// TIA Portal V19 export
// export: Created 2024-12-05T09:06:09.934265Z, ExportSetting WithDefaults, DisplayName Totally Integrated Automation Portal, DisplayVersion V19 Update 1, DisplayName TIA Portal Openness, DisplayVersion V19 Update 1, DisplayName TIA Portal Version Control Interface, DisplayVersion V19, DisplayName SINAMICS Startdrive Advanced, DisplayVersion V19, DisplayName SINAMICS DCC, DisplayVersion V19, DisplayName SINAMICS Startdrive G130, G150, S120, S150, SINAMICS MV, G220, S200, S210, DisplayVersion V19, DisplayName SINAMICS Startdrive G110M, G120, G120C, G120D, G120P, G115D, DisplayVersion V19, DisplayName STEP 7 Professional, DisplayVersion V19 Update 1, DisplayName STEP 7 Safety, DisplayVersion V19 Update 1, DisplayName WinCC Advanced, DisplayVersion V19 Update 1, DisplayName WinCC Advanced / Unified PC, DisplayVersion V19 Update 1
DATA_BLOCK "CH1"   // DB7
{ S7_Optimized_Access := 'TRUE' }
VERSION : 0.1
// stored: AutoNumber true, DBAccessibleFromOPCUA true, DBAccessibleFromWebserver true, InstanceOfName CH, InstanceOfType UDT, IsOnlyStoredInLoadMemory false, IsWriteProtectedInAS false
"CH"
   // VAR RETAIN
   //    Std : "EM_Std";
   //    Gen : "CH_Gen";
   //    Param : "CH_Param";
   //    LastHmiDataParam : "CH_Param";
   //    Alm : "CH_Alm";
   //    Sign : "EM_Sign";
   //    Input : "CH_Input";
   //    Output : "CH_Output";
   //    Ons : "CH_Ons";
   //    "Step" : "CH_Step";
   //    CamCalc : "CH_CamCalc";
   //    Chain1Long : "CH_Chain";
   //    Chain2Long : "CH_Chain";
   //    Chain3Long : "CH_Chain";
   //    Chain4Cross : "CH_Chain";
   //    Chain5Long : "CH_Chain";
   //    Chain6Long : "CH_Chain";
   //    Chain7Long : "CH_Chain";
   //    Chain8Cross : "CH_Chain";
   //    VMaster : "CH_Virtual";
   //    VMasterBooked : "CH_VirtualBooked";
   // END_VAR
BEGIN
   Std.Cfg_ModuleSync := TRUE;
   Std.Cfg_0_BelongShort_1_BelongLong := TRUE;
   Std.Cfg_ExternalCPU := FALSE;
   Std.Cfg_0_JogWord_1_JogBit := TRUE;
   Std._0_PriorityAlm_1_FirstAlm := FALSE;
   Std.AbortAlmOk := TRUE;
   Std.ServicesAbortAlmOk := FALSE;
   Std.SignOK := TRUE;
   Std.AlmReset := FALSE;
   Std.SignReset := FALSE;
   Std.NewAlm := FALSE;
   Std.NewSign := FALSE;
   Std.RstNewAlm := FALSE;
   Std.RstNewSign := FALSE;
   Std.AllowCopyByCategory := TRUE;
   Std.ForceCopyAll := FALSE;
   Std.InitCategories := FALSE;
   Std.InitCauses := FALSE;
   Std.Diag_AlmFound := FALSE;
   Std.Diag_SignFound := FALSE;
   Std.ScOk := FALSE;
   Std.OkToStop := TRUE;
   Std.PwrDrv := TRUE;
   Std.DriveRunCmd := FALSE;
   Std.ManAct := FALSE;
   Std.MachineSelected := TRUE;
   Std.MachineExtracted := FALSE;
   Std.LocalAbortReq := TRUE;
   Std.CondOkToEnaStaReq := FALSE;
   Std.EnaReq := FALSE;
   Std.EnaStaReq := FALSE;
   Std.StaReq := FALSE;
   Std.ReqStart := FALSE;
   Std.ReqStop := FALSE;
   Std.ReqAbort := TRUE;
   Std.ReqExecute := FALSE;
   Std.ReqReset := FALSE;
   Std.ReqSuspend := FALSE;
   Std.ReqUnSuspend := FALSE;
   Std.StrobeDeviceDiag := FALSE;
   Std.StrobeInverterDiag := FALSE;
   Std.DeviceDiagnosticDone := FALSE;
   Std.InverterDiagnosticDone := FALSE;
   Std.RecipeOnlineLoadDone := FALSE;
   Std.RecipeOnlineSaveDone := FALSE;
   Std.RecipeOfflineLoadDone := FALSE;
   Std.RecipeOfflineSaveDone := FALSE;
   Std.LastHmiDataLoadDone := FALSE;
   Std.LastHmiDataSaveDone := FALSE;
   Std.SummAlmTimeoutStart := FALSE;
   Std.SirenEna := FALSE;
   Std.VisEnButtons := TRUE;
   Std.VisManButtons := FALSE;
   Std.VisHomeButtons := FALSE;
   Std.VisEnButtonsRunning := TRUE;
   Std.Ena_Suspended := TRUE;
   Std.BluStkLgh_Steady_Cond := FALSE;
   Std.BluStkLgh_Frequency1_Cond := FALSE;
   Std.Siren_Frequency4_Cond := FALSE;
   Std.Cfg_ModuleNumber := 0;
   Std.Cfg_DeviceDiagCounter_Preset := 0;
   Std.Cfg_InverterDiagCounter_Preset := 0;
   Std.Cfg_Num_AlmDint := 19;
   Std.Cfg_Num_SignDint := 3;
   Std.Cfg_StaPbt := 65535;
   Std.Cfg_StoPbt := 65535;
   Std.Cfg_RstPbt := -1;
   Std.Cfg_EnaPbt := 65535;
   Std.Cfg_Siren := 1;
   Std.Cfg_Stack := 1;
   Std.Cfg_DisableStates[0..31] := 0;
   Std.Cfg_ModeTransitions[0..31] := 0;
   Std.Cfg_ModeNames[0..31] := '';
   Std.ModeCurrentName := 'Production';
   Std.StateCurrentName := 'Aborted';
   Std.DeviceDiagCounter := 0;
   Std.InverterDiagCounter := 0;
   Std.MaintenanceActivated."0" := FALSE;
   Std.MaintenanceActivated."1" := FALSE;
   Std.MaintenanceActivated."2" := FALSE;
   Std.MaintenanceActivated."3" := FALSE;
   Std.MaintenanceActivated."4" := FALSE;
   Std.MaintenanceActivated."5" := FALSE;
   Std.MaintenanceActivated."6" := FALSE;
   Std.MaintenanceActivated."7" := FALSE;
   Std.MaintenanceActivated."8" := FALSE;
   Std.MaintenanceActivated."9" := FALSE;
   Std.MaintenanceActivated."10" := FALSE;
   Std.MaintenanceActivated."11" := FALSE;
   Std.MaintenanceActivated."12" := FALSE;
   Std.MaintenanceActivated."13" := FALSE;
   Std.MaintenanceActivated."14" := FALSE;
   Std.MaintenanceActivated."15" := FALSE;
   Std.MaintenanceActivated."16" := FALSE;
   Std.MaintenanceActivated."17" := FALSE;
   Std.MaintenanceActivated."18" := FALSE;
   Std.MaintenanceActivated."19" := FALSE;
   Std.MaintenanceActivated."20" := FALSE;
   Std.MaintenanceActivated."21" := FALSE;
   Std.MaintenanceActivated."22" := FALSE;
   Std.MaintenanceActivated."23" := FALSE;
   Std.MaintenanceActivated."24" := FALSE;
   Std.MaintenanceActivated."25" := FALSE;
   Std.MaintenanceActivated."26" := FALSE;
   Std.MaintenanceActivated."27" := FALSE;
   Std.MaintenanceActivated."28" := FALSE;
   Std.MaintenanceActivated."29" := FALSE;
   Std.MaintenanceActivated."30" := FALSE;
   Std.MaintenanceActivated."31" := FALSE;
   Std.MaintenanceReq."0" := FALSE;
   Std.MaintenanceReq."1" := FALSE;
   Std.MaintenanceReq."2" := FALSE;
   Std.MaintenanceReq."3" := FALSE;
   Std.MaintenanceReq."4" := FALSE;
   Std.MaintenanceReq."5" := FALSE;
   Std.MaintenanceReq."6" := FALSE;
   Std.MaintenanceReq."7" := FALSE;
   Std.MaintenanceReq."8" := FALSE;
   Std.MaintenanceReq."9" := FALSE;
   Std.MaintenanceReq."10" := FALSE;
   Std.MaintenanceReq."11" := FALSE;
   Std.MaintenanceReq."12" := FALSE;
   Std.MaintenanceReq."13" := FALSE;
   Std.MaintenanceReq."14" := FALSE;
   Std.MaintenanceReq."15" := FALSE;
   Std.MaintenanceReq."16" := FALSE;
   Std.MaintenanceReq."17" := FALSE;
   Std.MaintenanceReq."18" := FALSE;
   Std.MaintenanceReq."19" := FALSE;
   Std.MaintenanceReq."20" := FALSE;
   Std.MaintenanceReq."21" := FALSE;
   Std.MaintenanceReq."22" := FALSE;
   Std.MaintenanceReq."23" := FALSE;
   Std.MaintenanceReq."24" := FALSE;
   Std.MaintenanceReq."25" := FALSE;
   Std.MaintenanceReq."26" := FALSE;
   Std.MaintenanceReq."27" := FALSE;
   Std.MaintenanceReq."28" := FALSE;
   Std.MaintenanceReq."29" := FALSE;
   Std.MaintenanceReq."30" := FALSE;
   Std.MaintenanceReq."31" := FALSE;
   Std.WithinScreenRange := 0;
   Std.ExchangeToGlobal.Communication.RunMode := FALSE;
   Std.ExchangeToGlobal.Communication.ConnectionFaulted := FALSE;
   Std.ExchangeToGlobal.Gen.Communication := FALSE;
   Std.ExchangeToGlobal.Gen.Selected := TRUE;
   Std.ExchangeToGlobal.Gen.Extracted := FALSE;
   Std.ExchangeToGlobal.Gen.EnaReq := FALSE;
   Std.ExchangeToGlobal.Gen.StaReq := FALSE;
   Std.ExchangeToGlobal.Gen.Started := FALSE;
   Std.ExchangeToGlobal.Gen.Unsuspended := FALSE;
   Std.ExchangeToGlobal.Gen.Ena_Suspended := TRUE;
   Std.ExchangeToGlobal.Gen.sts_Starting := FALSE;
   Std.ExchangeToGlobal.Gen.sts_Stopping := FALSE;
   Std.ExchangeToGlobal.Gen.sts_Aborting := FALSE;
   Std.ExchangeToGlobal.Gen.sts_Suspending := FALSE;
   Std.ExchangeToGlobal.Gen.sts_Unsuspending := FALSE;
   Std.ExchangeToGlobal.Gen.sts_Execute := FALSE;
   Std.ExchangeToGlobal.Gen.sts_Idle := FALSE;
   Std.ExchangeToGlobal.Gen.sts_Stopped := FALSE;
   Std.ExchangeToGlobal.Gen.sts_Aborted := TRUE;
   Std.ExchangeToGlobal.Gen.sts_Suspended := FALSE;
   Std.ExchangeToGlobal.Gen.sts_ModeManual := FALSE;
   Std.ExchangeToGlobal.Gen.sts_ModeAutomatic := TRUE;
   Std.ExchangeToGlobal.Gen.NewAlm := FALSE;
   Std.ExchangeToGlobal.Gen.NewSign := FALSE;
   Std.ExchangeToGlobal.Gen.RecipeOnlineLoadDone := FALSE;
   Std.ExchangeToGlobal.Gen.RecipeOnlineSaveDone := FALSE;
   Std.ExchangeToGlobal.Gen.RecipeOfflineLoadDone := FALSE;
   Std.ExchangeToGlobal.Gen.RecipeOfflineSaveDone := FALSE;
   Std.ExchangeToGlobal.Gen.LastHmiDataLoadDone := FALSE;
   Std.ExchangeToGlobal.Gen.LastHmiDataSaveDone := FALSE;
   Std.ExchangeToGlobal.Gen.InverterDiagnosticDone := FALSE;
   Std.ExchangeToGlobal.Gen.AxisGroupSync := TRUE;
   Std.ExchangeToGlobal.Gen.CmdMode := 1;
   Std.ExchangeToGlobal.Gen.Mode := 1;
   Std.ExchangeToGlobal.Gen.DisableEnaPbt := 0;
   Std.ExchangeToGlobal.Input.StaPbt := FALSE;
   Std.ExchangeToGlobal.Input.StoPbt := FALSE;
   Std.ExchangeToGlobal.Input.RstPbt := FALSE;
   Std.ExchangeToGlobal.Input.EnaPbt := FALSE;
   Std.ExchangeToGlobal.Input._4 := FALSE;
   Std.ExchangeToGlobal.Input._5 := FALSE;
   Std.ExchangeToGlobal.Input._6 := FALSE;
   Std.ExchangeToGlobal.Input._7 := FALSE;
   Std.ExchangeToGlobal.Input._8 := FALSE;
   Std.ExchangeToGlobal.Input._9 := FALSE;
   Std.ExchangeToGlobal.Input._10 := FALSE;
   Std.ExchangeToGlobal.Input._11 := FALSE;
   Std.ExchangeToGlobal.Input._12 := FALSE;
   Std.ExchangeToGlobal.Input._13 := FALSE;
   Std.ExchangeToGlobal.Input._14 := FALSE;
   Std.ExchangeToGlobal.Input._15 := FALSE;
   Std.ExchangeToGlobal.AlmOk.ThSwitch := TRUE;
   Std.ExchangeToGlobal.AlmOk.SafeComm := TRUE;
   Std.ExchangeToGlobal.AlmOk.SafeEmg := TRUE;
   Std.ExchangeToGlobal.AlmOk.SafeGuards := TRUE;
   Std.ExchangeToGlobal.AlmOk.GtaAirGroup := TRUE;
   Std.ExchangeToGlobal.AlmOk.Major := TRUE;
   Std.ExchangeToGlobal.AlmOk.Minor := TRUE;
   Std.ExchangeToGlobal.AlmOk.Spare07 := TRUE;
   Std.ExchangeToGlobal.AlmOk.Spare08 := TRUE;
   Std.ExchangeToGlobal.AlmOk.Spare09 := TRUE;
   Std.ExchangeToGlobal.AlmOk.Spare10 := TRUE;
   Std.ExchangeToGlobal.AlmOk.Spare11 := TRUE;
   Std.ExchangeToGlobal.AlmOk.Spare12 := TRUE;
   Std.ExchangeToGlobal.AlmOk.Spare13 := TRUE;
   Std.ExchangeToGlobal.AlmOk.Spare14 := TRUE;
   Std.ExchangeToGlobal.AlmOk.Spare15 := TRUE;
   Std.ExchangeToGlobal.AlmOk.Spare16 := TRUE;
   Std.ExchangeToGlobal.AlmOk.Spare17 := TRUE;
   Std.ExchangeToGlobal.AlmOk.Spare18 := TRUE;
   Std.ExchangeToGlobal.AlmOk.Spare19 := TRUE;
   Std.ExchangeToGlobal.AlmOk.Spare20 := TRUE;
   Std.ExchangeToGlobal.AlmOk.Spare21 := TRUE;
   Std.ExchangeToGlobal.AlmOk.Spare22 := TRUE;
   Std.ExchangeToGlobal.AlmOk.Spare23 := TRUE;
   Std.ExchangeToGlobal.AlmOk.Spare24 := TRUE;
   Std.ExchangeToGlobal.AlmOk.Spare25 := TRUE;
   Std.ExchangeToGlobal.AlmOk.Spare26 := TRUE;
   Std.ExchangeToGlobal.AlmOk.Spare27 := TRUE;
   Std.ExchangeToGlobal.AlmOk.Spare28 := TRUE;
   Std.ExchangeToGlobal.AlmOk.Spare29 := TRUE;
   Std.ExchangeToGlobal.AlmOk.Spare30 := TRUE;
   Std.ExchangeToGlobal.AlmOk.Spare31 := TRUE;
   Std.ExchangeToGlobal.AlmCauseOk.Ope := TRUE;
   Std.ExchangeToGlobal.AlmCauseOk.Ust := TRUE;
   Std.ExchangeToGlobal.AlmCauseOk.Dst := TRUE;
   Std.ExchangeToGlobal.AlmCauseOk.Ext := TRUE;
   Std.ExchangeToGlobal.AlmCauseOk.Mac := TRUE;
   Std.ExchangeToGlobal.AlmCauseOk.Spare05 := TRUE;
   Std.ExchangeToGlobal.AlmCauseOk.Spare06 := TRUE;
   Std.ExchangeToGlobal.AlmCauseOk.Spare07 := TRUE;
   Std.ExchangeToGlobal.AlmCauseOk.Spare08 := TRUE;
   Std.ExchangeToGlobal.AlmCauseOk.Spare09 := TRUE;
   Std.ExchangeToGlobal.AlmCauseOk.Spare10 := TRUE;
   Std.ExchangeToGlobal.AlmCauseOk.Spare11 := TRUE;
   Std.ExchangeToGlobal.AlmCauseOk.Spare12 := TRUE;
   Std.ExchangeToGlobal.AlmCauseOk.Spare13 := TRUE;
   Std.ExchangeToGlobal.AlmCauseOk.Spare14 := TRUE;
   Std.ExchangeToGlobal.AlmCauseOk.Spare15 := TRUE;
   Std.ExchangeToGlobal.AlmCauseOk.Spare16 := TRUE;
   Std.ExchangeToGlobal.AlmCauseOk.Spare17 := TRUE;
   Std.ExchangeToGlobal.AlmCauseOk.Spare18 := TRUE;
   Std.ExchangeToGlobal.AlmCauseOk.Spare19 := TRUE;
   Std.ExchangeToGlobal.AlmCauseOk.Spare20 := TRUE;
   Std.ExchangeToGlobal.AlmCauseOk.Spare21 := TRUE;
   Std.ExchangeToGlobal.AlmCauseOk.Spare22 := TRUE;
   Std.ExchangeToGlobal.AlmCauseOk.Spare23 := TRUE;
   Std.ExchangeToGlobal.AlmCauseOk.Spare24 := TRUE;
   Std.ExchangeToGlobal.AlmCauseOk.Spare25 := TRUE;
   Std.ExchangeToGlobal.AlmCauseOk.Spare26 := TRUE;
   Std.ExchangeToGlobal.AlmCauseOk.Spare27 := TRUE;
   Std.ExchangeToGlobal.AlmCauseOk.Spare28 := TRUE;
   Std.ExchangeToGlobal.AlmCauseOk.Spare29 := TRUE;
   Std.ExchangeToGlobal.AlmCauseOk.Spare30 := TRUE;
   Std.ExchangeToGlobal.AlmCauseOk.Spare31 := TRUE;
   Std.ExchangeToGlobal.AlmBannerFbk.FirstAlmDetection := FALSE;
   Std.ExchangeToGlobal.AlmBannerFbk.AlmPriority := 100;
   Std.ExchangeToGlobal.AlmBannerFbk.AlmCategory := -1;
   Std.ExchangeToGlobal.AlmBannerFbk.AlmCause := -1;
   Std.ExchangeToGlobal.AlmBannerFbk.AlmID := -1;
   Std.ExchangeToGlobal.AlmBannerFbk.GlobalAbsTime := 0;
   Std.ExchangeToGlobal.SignBannerFbk.SignPriority := 100;
   Std.ExchangeToGlobal.SignBannerFbk.SignCategory := -1;
   Std.ExchangeToGlobal.SignBannerFbk.SignID := -1;
   Std.ExchangeToGlobal.ExtCPU.PushButton.StaPbt := FALSE;
   Std.ExchangeToGlobal.ExtCPU.PushButton.StoPbt := FALSE;
   Std.ExchangeToGlobal.ExtCPU.PushButton.RstPbt := FALSE;
   Std.ExchangeToGlobal.ExtCPU.PushButton.EnaPbt := FALSE;
   Std.ExchangeToGlobal.ExtCPU.PushButton.EnaReq := FALSE;
   Std.ExchangeToGlobal.ExtCPU.PushButton.EnaStaReq := FALSE;
   Std.ExchangeToGlobal.ExtCPU.DeviceDiagDone := FALSE;
   Std.ExchangeToGlobal.ExtCPU.InverterDiagDone := FALSE;
   Std.ExchangeToGlobal.LightSiren.Cfg_StaPbt := 65535;
   Std.ExchangeToGlobal.LightSiren.Cfg_RstPbt := -1;
   Std.ExchangeToGlobal.LightSiren.Cfg_EnaPbt := 65535;
   Std.ExchangeToGlobal.LightSiren.Cfg_Siren := 1;
   Std.ExchangeToGlobal.LightSiren.Cfg_Stack := 1;
   Std.ExchangeToGlobal.LightSiren.Steady.StaPbtLgh := FALSE;
   Std.ExchangeToGlobal.LightSiren.Steady.RstPbtLgh := FALSE;
   Std.ExchangeToGlobal.LightSiren.Steady.EnaPbtLgh := FALSE;
   Std.ExchangeToGlobal.LightSiren.Steady.Siren := FALSE;
   Std.ExchangeToGlobal.LightSiren.Steady.YelStkLgh := FALSE;
   Std.ExchangeToGlobal.LightSiren.Steady.BluStkLgh := FALSE;
   Std.ExchangeToGlobal.LightSiren.Steady.GrnStkLgh := FALSE;
   Std.ExchangeToGlobal.LightSiren.Steady.WhtStkLgh := FALSE;
   Std.ExchangeToGlobal.LightSiren.Steady.Cust1_StaPbtLgh := FALSE;
   Std.ExchangeToGlobal.LightSiren.Steady.Cust1_RstPbtLgh := FALSE;
   Std.ExchangeToGlobal.LightSiren.Steady.Cust1_Siren := FALSE;
   Std.ExchangeToGlobal.LightSiren.Steady.Cust1_RedStkLgh := FALSE;
   Std.ExchangeToGlobal.LightSiren.Steady.Cust1_OngStkLgh := FALSE;
   Std.ExchangeToGlobal.LightSiren.Steady.Cust1_GrnStkLgh := FALSE;
   Std.ExchangeToGlobal.LightSiren.Steady.Cust1_BluStkLgh := FALSE;
   Std.ExchangeToGlobal.LightSiren.Steady.Cust1_WhtStkLgh := FALSE;
   Std.ExchangeToGlobal.LightSiren.Frequency1.StaPbtLgh := FALSE;
   Std.ExchangeToGlobal.LightSiren.Frequency1.RstPbtLgh := FALSE;
   Std.ExchangeToGlobal.LightSiren.Frequency1.EnaPbtLgh := FALSE;
   Std.ExchangeToGlobal.LightSiren.Frequency1.Siren := FALSE;
   Std.ExchangeToGlobal.LightSiren.Frequency1.YelStkLgh := FALSE;
   Std.ExchangeToGlobal.LightSiren.Frequency1.BluStkLgh := FALSE;
   Std.ExchangeToGlobal.LightSiren.Frequency1.GrnStkLgh := FALSE;
   Std.ExchangeToGlobal.LightSiren.Frequency1.WhtStkLgh := FALSE;
   Std.ExchangeToGlobal.LightSiren.Frequency1.Cust1_StaPbtLgh := FALSE;
   Std.ExchangeToGlobal.LightSiren.Frequency1.Cust1_RstPbtLgh := FALSE;
   Std.ExchangeToGlobal.LightSiren.Frequency1.Cust1_Siren := FALSE;
   Std.ExchangeToGlobal.LightSiren.Frequency1.Cust1_RedStkLgh := FALSE;
   Std.ExchangeToGlobal.LightSiren.Frequency1.Cust1_OngStkLgh := FALSE;
   Std.ExchangeToGlobal.LightSiren.Frequency1.Cust1_GrnStkLgh := FALSE;
   Std.ExchangeToGlobal.LightSiren.Frequency1.Cust1_BluStkLgh := FALSE;
   Std.ExchangeToGlobal.LightSiren.Frequency1.Cust1_WhtStkLgh := FALSE;
   Std.ExchangeToGlobal.LightSiren.Frequency2.StaPbtLgh := FALSE;
   Std.ExchangeToGlobal.LightSiren.Frequency2.RstPbtLgh := FALSE;
   Std.ExchangeToGlobal.LightSiren.Frequency2.EnaPbtLgh := FALSE;
   Std.ExchangeToGlobal.LightSiren.Frequency2.Siren := FALSE;
   Std.ExchangeToGlobal.LightSiren.Frequency2.YelStkLgh := FALSE;
   Std.ExchangeToGlobal.LightSiren.Frequency2.BluStkLgh := FALSE;
   Std.ExchangeToGlobal.LightSiren.Frequency2.GrnStkLgh := FALSE;
   Std.ExchangeToGlobal.LightSiren.Frequency2.WhtStkLgh := FALSE;
   Std.ExchangeToGlobal.LightSiren.Frequency2.Cust1_StaPbtLgh := FALSE;
   Std.ExchangeToGlobal.LightSiren.Frequency2.Cust1_RstPbtLgh := FALSE;
   Std.ExchangeToGlobal.LightSiren.Frequency2.Cust1_Siren := FALSE;
   Std.ExchangeToGlobal.LightSiren.Frequency2.Cust1_RedStkLgh := FALSE;
   Std.ExchangeToGlobal.LightSiren.Frequency2.Cust1_OngStkLgh := FALSE;
   Std.ExchangeToGlobal.LightSiren.Frequency2.Cust1_GrnStkLgh := FALSE;
   Std.ExchangeToGlobal.LightSiren.Frequency2.Cust1_BluStkLgh := FALSE;
   Std.ExchangeToGlobal.LightSiren.Frequency2.Cust1_WhtStkLgh := FALSE;
   Std.ExchangeToGlobal.LightSiren.Frequency3.StaPbtLgh := FALSE;
   Std.ExchangeToGlobal.LightSiren.Frequency3.RstPbtLgh := FALSE;
   Std.ExchangeToGlobal.LightSiren.Frequency3.EnaPbtLgh := FALSE;
   Std.ExchangeToGlobal.LightSiren.Frequency3.Siren := FALSE;
   Std.ExchangeToGlobal.LightSiren.Frequency3.YelStkLgh := FALSE;
   Std.ExchangeToGlobal.LightSiren.Frequency3.BluStkLgh := FALSE;
   Std.ExchangeToGlobal.LightSiren.Frequency3.GrnStkLgh := FALSE;
   Std.ExchangeToGlobal.LightSiren.Frequency3.WhtStkLgh := FALSE;
   Std.ExchangeToGlobal.LightSiren.Frequency3.Cust1_StaPbtLgh := FALSE;
   Std.ExchangeToGlobal.LightSiren.Frequency3.Cust1_RstPbtLgh := FALSE;
   Std.ExchangeToGlobal.LightSiren.Frequency3.Cust1_Siren := FALSE;
   Std.ExchangeToGlobal.LightSiren.Frequency3.Cust1_RedStkLgh := FALSE;
   Std.ExchangeToGlobal.LightSiren.Frequency3.Cust1_OngStkLgh := FALSE;
   Std.ExchangeToGlobal.LightSiren.Frequency3.Cust1_GrnStkLgh := FALSE;
   Std.ExchangeToGlobal.LightSiren.Frequency3.Cust1_BluStkLgh := FALSE;
   Std.ExchangeToGlobal.LightSiren.Frequency3.Cust1_WhtStkLgh := FALSE;
   Std.ExchangeToGlobal.LightSiren.Frequency4.StaPbtLgh := FALSE;
   Std.ExchangeToGlobal.LightSiren.Frequency4.RstPbtLgh := FALSE;
   Std.ExchangeToGlobal.LightSiren.Frequency4.EnaPbtLgh := FALSE;
   Std.ExchangeToGlobal.LightSiren.Frequency4.Siren := FALSE;
   Std.ExchangeToGlobal.LightSiren.Frequency4.YelStkLgh := FALSE;
   Std.ExchangeToGlobal.LightSiren.Frequency4.BluStkLgh := FALSE;
   Std.ExchangeToGlobal.LightSiren.Frequency4.GrnStkLgh := FALSE;
   Std.ExchangeToGlobal.LightSiren.Frequency4.WhtStkLgh := FALSE;
   Std.ExchangeToGlobal.LightSiren.Frequency4.Cust1_StaPbtLgh := FALSE;
   Std.ExchangeToGlobal.LightSiren.Frequency4.Cust1_RstPbtLgh := FALSE;
   Std.ExchangeToGlobal.LightSiren.Frequency4.Cust1_Siren := FALSE;
   Std.ExchangeToGlobal.LightSiren.Frequency4.Cust1_RedStkLgh := FALSE;
   Std.ExchangeToGlobal.LightSiren.Frequency4.Cust1_OngStkLgh := FALSE;
   Std.ExchangeToGlobal.LightSiren.Frequency4.Cust1_GrnStkLgh := FALSE;
   Std.ExchangeToGlobal.LightSiren.Frequency4.Cust1_BluStkLgh := FALSE;
   Std.ExchangeToGlobal.LightSiren.Frequency4.Cust1_WhtStkLgh := FALSE;
   Std.ExchangeToGlobal.PackML.Sts_Aborted := TRUE;
   Std.ExchangeToGlobal.PackML.Sts_Aborting := FALSE;
   Std.ExchangeToGlobal.PackML.Sts_Clearing := FALSE;
   Std.ExchangeToGlobal.PackML.Sts_Complete := FALSE;
   Std.ExchangeToGlobal.PackML.Sts_Completing := FALSE;
   Std.ExchangeToGlobal.PackML.Sts_Execute := FALSE;
   Std.ExchangeToGlobal.PackML.Sts_Held := FALSE;
   Std.ExchangeToGlobal.PackML.Sts_Holding := FALSE;
   Std.ExchangeToGlobal.PackML.Sts_Idle := FALSE;
   Std.ExchangeToGlobal.PackML.Sts_Resetting := FALSE;
   Std.ExchangeToGlobal.PackML.Sts_Starting := FALSE;
   Std.ExchangeToGlobal.PackML.Sts_Stopped := FALSE;
   Std.ExchangeToGlobal.PackML.Sts_Stopping := FALSE;
   Std.ExchangeToGlobal.PackML.Sts_Suspended := FALSE;
   Std.ExchangeToGlobal.PackML.Sts_Suspending := FALSE;
   Std.ExchangeToGlobal.PackML.Sts_UnHolding := FALSE;
   Std.ExchangeToGlobal.PackML.Sts_UnSuspending := FALSE;
   Std.ExchangeToGlobal.PackML.Sts_AbortedEnabled := TRUE;
   Std.ExchangeToGlobal.PackML.Sts_AbortingEnabled := TRUE;
   Std.ExchangeToGlobal.PackML.Sts_ClearingEnabled := TRUE;
   Std.ExchangeToGlobal.PackML.Sts_CompleteEnabled := FALSE;
   Std.ExchangeToGlobal.PackML.Sts_CompletingEnabled := FALSE;
   Std.ExchangeToGlobal.PackML.Sts_ExecuteEnabled := TRUE;
   Std.ExchangeToGlobal.PackML.Sts_HeldEnabled := FALSE;
   Std.ExchangeToGlobal.PackML.Sts_HoldingEnabled := FALSE;
   Std.ExchangeToGlobal.PackML.Sts_IdleEnabled := TRUE;
   Std.ExchangeToGlobal.PackML.Sts_ResettingEnabled := TRUE;
   Std.ExchangeToGlobal.PackML.Sts_StartingEnabled := TRUE;
   Std.ExchangeToGlobal.PackML.Sts_StoppedEnabled := TRUE;
   Std.ExchangeToGlobal.PackML.Sts_StoppingEnabled := TRUE;
   Std.ExchangeToGlobal.PackML.Sts_SuspendedEnabled := TRUE;
   Std.ExchangeToGlobal.PackML.Sts_SuspendingEnabled := TRUE;
   Std.ExchangeToGlobal.PackML.Sts_UnHoldingEnabled := FALSE;
   Std.ExchangeToGlobal.PackML.Sts_UnSuspendingEnabled := TRUE;
   Std.ExchangeToGlobal.SignOk := TRUE;
   Std.ExchangeToGlobal."Dint"[0..4] := 0;
   Std.VisAlmTypeBool.ThSwitch := FALSE;
   Std.VisAlmTypeBool.SafeComm := FALSE;
   Std.VisAlmTypeBool.SafeEmg := FALSE;
   Std.VisAlmTypeBool.SafeGuards := TRUE;
   Std.VisAlmTypeBool.GtaAirGroup := FALSE;
   Std.VisAlmTypeBool.Major := FALSE;
   Std.VisAlmTypeBool.Minor := FALSE;
   Std.VisAlmTypeBool.Spare07 := FALSE;
   Std.VisAlmTypeBool.Spare08 := FALSE;
   Std.VisAlmTypeBool.Spare09 := FALSE;
   Std.VisAlmTypeBool.Spare10 := FALSE;
   Std.VisAlmTypeBool.Spare11 := FALSE;
   Std.VisAlmTypeBool.Spare12 := FALSE;
   Std.VisAlmTypeBool.Spare13 := FALSE;
   Std.VisAlmTypeBool.Spare14 := FALSE;
   Std.VisAlmTypeBool.Spare15 := FALSE;
   Std.VisAlmTypeBool.Spare16 := FALSE;
   Std.VisAlmTypeBool.Spare17 := FALSE;
   Std.VisAlmTypeBool.Spare18 := FALSE;
   Std.VisAlmTypeBool.Spare19 := FALSE;
   Std.VisAlmTypeBool.Spare20 := FALSE;
   Std.VisAlmTypeBool.Spare21 := FALSE;
   Std.VisAlmTypeBool.Spare22 := FALSE;
   Std.VisAlmTypeBool.Spare23 := FALSE;
   Std.VisAlmTypeBool.Spare24 := FALSE;
   Std.VisAlmTypeBool.Spare25 := FALSE;
   Std.VisAlmTypeBool.Spare26 := FALSE;
   Std.VisAlmTypeBool.Spare27 := FALSE;
   Std.VisAlmTypeBool.Spare28 := FALSE;
   Std.VisAlmTypeBool.Spare29 := FALSE;
   Std.VisAlmTypeBool.Spare30 := FALSE;
   Std.VisAlmTypeBool.Spare31 := FALSE;
   Std.AlmTypeFbk.ThSwitch := FALSE;
   Std.AlmTypeFbk.SafeComm := FALSE;
   Std.AlmTypeFbk.SafeEmg := FALSE;
   Std.AlmTypeFbk.SafeGuards := FALSE;
   Std.AlmTypeFbk.GtaAirGroup := FALSE;
   Std.AlmTypeFbk.Major := FALSE;
   Std.AlmTypeFbk.Minor := FALSE;
   Std.AlmTypeFbk.Spare07 := FALSE;
   Std.AlmTypeFbk.Spare08 := FALSE;
   Std.AlmTypeFbk.Spare09 := FALSE;
   Std.AlmTypeFbk.Spare10 := FALSE;
   Std.AlmTypeFbk.Spare11 := FALSE;
   Std.AlmTypeFbk.Spare12 := FALSE;
   Std.AlmTypeFbk.Spare13 := FALSE;
   Std.AlmTypeFbk.Spare14 := FALSE;
   Std.AlmTypeFbk.Spare15 := FALSE;
   Std.AlmTypeFbk.Spare16 := FALSE;
   Std.AlmTypeFbk.Spare17 := FALSE;
   Std.AlmTypeFbk.Spare18 := FALSE;
   Std.AlmTypeFbk.Spare19 := FALSE;
   Std.AlmTypeFbk.Spare20 := FALSE;
   Std.AlmTypeFbk.Spare21 := FALSE;
   Std.AlmTypeFbk.Spare22 := FALSE;
   Std.AlmTypeFbk.Spare23 := FALSE;
   Std.AlmTypeFbk.Spare24 := FALSE;
   Std.AlmTypeFbk.Spare25 := FALSE;
   Std.AlmTypeFbk.Spare26 := FALSE;
   Std.AlmTypeFbk.Spare27 := FALSE;
   Std.AlmTypeFbk.Spare28 := FALSE;
   Std.AlmTypeFbk.Spare29 := FALSE;
   Std.AlmTypeFbk.Spare30 := FALSE;
   Std.AlmTypeFbk.Spare31 := FALSE;
   Std.AlmTypeOk.ThSwitch := TRUE;
   Std.AlmTypeOk.SafeComm := TRUE;
   Std.AlmTypeOk.SafeEmg := TRUE;
   Std.AlmTypeOk.SafeGuards := TRUE;
   Std.AlmTypeOk.GtaAirGroup := TRUE;
   Std.AlmTypeOk.Major := TRUE;
   Std.AlmTypeOk.Minor := TRUE;
   Std.AlmTypeOk.Spare07 := TRUE;
   Std.AlmTypeOk.Spare08 := TRUE;
   Std.AlmTypeOk.Spare09 := TRUE;
   Std.AlmTypeOk.Spare10 := TRUE;
   Std.AlmTypeOk.Spare11 := TRUE;
   Std.AlmTypeOk.Spare12 := TRUE;
   Std.AlmTypeOk.Spare13 := TRUE;
   Std.AlmTypeOk.Spare14 := TRUE;
   Std.AlmTypeOk.Spare15 := TRUE;
   Std.AlmTypeOk.Spare16 := TRUE;
   Std.AlmTypeOk.Spare17 := TRUE;
   Std.AlmTypeOk.Spare18 := TRUE;
   Std.AlmTypeOk.Spare19 := TRUE;
   Std.AlmTypeOk.Spare20 := TRUE;
   Std.AlmTypeOk.Spare21 := TRUE;
   Std.AlmTypeOk.Spare22 := TRUE;
   Std.AlmTypeOk.Spare23 := TRUE;
   Std.AlmTypeOk.Spare24 := TRUE;
   Std.AlmTypeOk.Spare25 := TRUE;
   Std.AlmTypeOk.Spare26 := TRUE;
   Std.AlmTypeOk.Spare27 := TRUE;
   Std.AlmTypeOk.Spare28 := TRUE;
   Std.AlmTypeOk.Spare29 := TRUE;
   Std.AlmTypeOk.Spare30 := TRUE;
   Std.AlmTypeOk.Spare31 := TRUE;
   Std.AlmCauseFbk.Ope := FALSE;
   Std.AlmCauseFbk.Ust := FALSE;
   Std.AlmCauseFbk.Dst := FALSE;
   Std.AlmCauseFbk.Ext := FALSE;
   Std.AlmCauseFbk.Mac := FALSE;
   Std.AlmCauseFbk.Spare05 := FALSE;
   Std.AlmCauseFbk.Spare06 := FALSE;
   Std.AlmCauseFbk.Spare07 := FALSE;
   Std.AlmCauseFbk.Spare08 := FALSE;
   Std.AlmCauseFbk.Spare09 := FALSE;
   Std.AlmCauseFbk.Spare10 := FALSE;
   Std.AlmCauseFbk.Spare11 := FALSE;
   Std.AlmCauseFbk.Spare12 := FALSE;
   Std.AlmCauseFbk.Spare13 := FALSE;
   Std.AlmCauseFbk.Spare14 := FALSE;
   Std.AlmCauseFbk.Spare15 := FALSE;
   Std.AlmCauseFbk.Spare16 := FALSE;
   Std.AlmCauseFbk.Spare17 := FALSE;
   Std.AlmCauseFbk.Spare18 := FALSE;
   Std.AlmCauseFbk.Spare19 := FALSE;
   Std.AlmCauseFbk.Spare20 := FALSE;
   Std.AlmCauseFbk.Spare21 := FALSE;
   Std.AlmCauseFbk.Spare22 := FALSE;
   Std.AlmCauseFbk.Spare23 := FALSE;
   Std.AlmCauseFbk.Spare24 := FALSE;
   Std.AlmCauseFbk.Spare25 := FALSE;
   Std.AlmCauseFbk.Spare26 := FALSE;
   Std.AlmCauseFbk.Spare27 := FALSE;
   Std.AlmCauseFbk.Spare28 := FALSE;
   Std.AlmCauseFbk.Spare29 := FALSE;
   Std.AlmCauseFbk.Spare30 := FALSE;
   Std.AlmCauseFbk.Spare31 := FALSE;
   Std.AlmCauseOk.Ope := TRUE;
   Std.AlmCauseOk.Ust := TRUE;
   Std.AlmCauseOk.Dst := TRUE;
   Std.AlmCauseOk.Ext := TRUE;
   Std.AlmCauseOk.Mac := TRUE;
   Std.AlmCauseOk.Spare05 := TRUE;
   Std.AlmCauseOk.Spare06 := TRUE;
   Std.AlmCauseOk.Spare07 := TRUE;
   Std.AlmCauseOk.Spare08 := TRUE;
   Std.AlmCauseOk.Spare09 := TRUE;
   Std.AlmCauseOk.Spare10 := TRUE;
   Std.AlmCauseOk.Spare11 := TRUE;
   Std.AlmCauseOk.Spare12 := TRUE;
   Std.AlmCauseOk.Spare13 := TRUE;
   Std.AlmCauseOk.Spare14 := TRUE;
   Std.AlmCauseOk.Spare15 := TRUE;
   Std.AlmCauseOk.Spare16 := TRUE;
   Std.AlmCauseOk.Spare17 := TRUE;
   Std.AlmCauseOk.Spare18 := TRUE;
   Std.AlmCauseOk.Spare19 := TRUE;
   Std.AlmCauseOk.Spare20 := TRUE;
   Std.AlmCauseOk.Spare21 := TRUE;
   Std.AlmCauseOk.Spare22 := TRUE;
   Std.AlmCauseOk.Spare23 := TRUE;
   Std.AlmCauseOk.Spare24 := TRUE;
   Std.AlmCauseOk.Spare25 := TRUE;
   Std.AlmCauseOk.Spare26 := TRUE;
   Std.AlmCauseOk.Spare27 := TRUE;
   Std.AlmCauseOk.Spare28 := TRUE;
   Std.AlmCauseOk.Spare29 := TRUE;
   Std.AlmCauseOk.Spare30 := TRUE;
   Std.AlmCauseOk.Spare31 := TRUE;
   Std.ForceCategory.ThSwitch := FALSE;
   Std.ForceCategory.SafeComm := TRUE;
   Std.ForceCategory.SafeEmg := TRUE;
   Std.ForceCategory.SafeGuards := FALSE;
   Std.ForceCategory.GtaAirGroup := FALSE;
   Std.ForceCategory.Major := FALSE;
   Std.ForceCategory.Minor := FALSE;
   Std.ForceCategory.Spare07 := FALSE;
   Std.ForceCategory.Spare08 := FALSE;
   Std.ForceCategory.Spare09 := FALSE;
   Std.ForceCategory.Spare10 := FALSE;
   Std.ForceCategory.Spare11 := FALSE;
   Std.ForceCategory.Spare12 := FALSE;
   Std.ForceCategory.Spare13 := FALSE;
   Std.ForceCategory.Spare14 := FALSE;
   Std.ForceCategory.Spare15 := FALSE;
   Std.ForceCategory.Spare16 := FALSE;
   Std.ForceCategory.Spare17 := FALSE;
   Std.ForceCategory.Spare18 := FALSE;
   Std.ForceCategory.Spare19 := FALSE;
   Std.ForceCategory.Spare20 := FALSE;
   Std.ForceCategory.Spare21 := FALSE;
   Std.ForceCategory.Spare22 := FALSE;
   Std.ForceCategory.Spare23 := FALSE;
   Std.ForceCategory.Spare24 := FALSE;
   Std.ForceCategory.Spare25 := FALSE;
   Std.ForceCategory.Spare26 := FALSE;
   Std.ForceCategory.Spare27 := FALSE;
   Std.ForceCategory.Spare28 := FALSE;
   Std.ForceCategory.Spare29 := FALSE;
   Std.ForceCategory.Spare30 := FALSE;
   Std.ForceCategory.Spare31 := FALSE;
   Std.AlmStruct.Alm[0..31] := 0;
   Std.AlmStruct.Category[0..31] := 0;
   Std.AlmStruct.Category[32..63] := 1;
   Std.AlmStruct.Category[64..95] := 2;
   Std.AlmStruct.Category[96..127] := 3;
   Std.AlmStruct.Category[128..159] := 4;
   Std.AlmStruct.Category[160..191] := 5;
   Std.AlmStruct.Category[192..1023] := 6;
   Std.AlmStruct.BannerPriority[0..31] := 0;
   Std.AlmStruct.BannerPriority[32..63] := 1;
   Std.AlmStruct.BannerPriority[64..95] := 2;
   Std.AlmStruct.BannerPriority[96..127] := 3;
   Std.AlmStruct.BannerPriority[128..159] := 4;
   Std.AlmStruct.BannerPriority[160..191] := 5;
   Std.AlmStruct.BannerPriority[192..1023] := 6;
   Std.AlmStruct.Cause[0..63] := 4;
   Std.AlmStruct.Cause[64..127] := 0;
   Std.AlmStruct.Cause[128..159] := 3;
   Std.AlmStruct.Cause[160..1023] := 4;
   Std.AlmBannerFbk.FirstAlmDetection := FALSE;
   Std.AlmBannerFbk.AlmPriority := 100;
   Std.AlmBannerFbk.AlmCategory := -1;
   Std.AlmBannerFbk.AlmCause := -1;
   Std.AlmBannerFbk.AlmID := -1;
   Std.AlmBannerFbk.GlobalAbsTime := 0;
   Std.SignStruct.Sign[0..31] := 0;
   Std.SignStruct.Category[0..1023] := 0;
   Std.SignStruct.BannerPriority[0..31] := 3;
   Std.SignStruct.BannerPriority[32..63] := 1;
   Std.SignStruct.BannerPriority[64..95] := 2;
   Std.SignStruct.BannerPriority[96..1023] := 0;
   Std.SignBannerFbk.SignPriority := 100;
   Std.SignBannerFbk.SignCategory := -1;
   Std.SignBannerFbk.SignID := -1;
   Std.MaintenanceInput.Clock_1Hz := FALSE;
   Std.MaintenanceInput.CountEnable := FALSE;
   Std.MaintenanceInput.CondToBeActivated := TRUE;
   Std.MaintenanceInput.EventsStrobe := 0;
   Std.LightSiren.Cfg_StaPbt := 65535;
   Std.LightSiren.Cfg_RstPbt := -1;
   Std.LightSiren.Cfg_EnaPbt := 65535;
   Std.LightSiren.Cfg_Siren := 1;
   Std.LightSiren.Cfg_Stack := 1;
   Std.LightSiren.Steady.StaPbtLgh := FALSE;
   Std.LightSiren.Steady.RstPbtLgh := FALSE;
   Std.LightSiren.Steady.EnaPbtLgh := FALSE;
   Std.LightSiren.Steady.Siren := FALSE;
   Std.LightSiren.Steady.YelStkLgh := FALSE;
   Std.LightSiren.Steady.BluStkLgh := FALSE;
   Std.LightSiren.Steady.GrnStkLgh := FALSE;
   Std.LightSiren.Steady.WhtStkLgh := FALSE;
   Std.LightSiren.Steady.Cust1_StaPbtLgh := FALSE;
   Std.LightSiren.Steady.Cust1_RstPbtLgh := FALSE;
   Std.LightSiren.Steady.Cust1_Siren := FALSE;
   Std.LightSiren.Steady.Cust1_RedStkLgh := FALSE;
   Std.LightSiren.Steady.Cust1_OngStkLgh := FALSE;
   Std.LightSiren.Steady.Cust1_GrnStkLgh := FALSE;
   Std.LightSiren.Steady.Cust1_BluStkLgh := FALSE;
   Std.LightSiren.Steady.Cust1_WhtStkLgh := FALSE;
   Std.LightSiren.Frequency1.StaPbtLgh := FALSE;
   Std.LightSiren.Frequency1.RstPbtLgh := FALSE;
   Std.LightSiren.Frequency1.EnaPbtLgh := FALSE;
   Std.LightSiren.Frequency1.Siren := FALSE;
   Std.LightSiren.Frequency1.YelStkLgh := FALSE;
   Std.LightSiren.Frequency1.BluStkLgh := FALSE;
   Std.LightSiren.Frequency1.GrnStkLgh := FALSE;
   Std.LightSiren.Frequency1.WhtStkLgh := FALSE;
   Std.LightSiren.Frequency1.Cust1_StaPbtLgh := FALSE;
   Std.LightSiren.Frequency1.Cust1_RstPbtLgh := FALSE;
   Std.LightSiren.Frequency1.Cust1_Siren := FALSE;
   Std.LightSiren.Frequency1.Cust1_RedStkLgh := FALSE;
   Std.LightSiren.Frequency1.Cust1_OngStkLgh := FALSE;
   Std.LightSiren.Frequency1.Cust1_GrnStkLgh := FALSE;
   Std.LightSiren.Frequency1.Cust1_BluStkLgh := FALSE;
   Std.LightSiren.Frequency1.Cust1_WhtStkLgh := FALSE;
   Std.LightSiren.Frequency2.StaPbtLgh := FALSE;
   Std.LightSiren.Frequency2.RstPbtLgh := FALSE;
   Std.LightSiren.Frequency2.EnaPbtLgh := FALSE;
   Std.LightSiren.Frequency2.Siren := FALSE;
   Std.LightSiren.Frequency2.YelStkLgh := FALSE;
   Std.LightSiren.Frequency2.BluStkLgh := FALSE;
   Std.LightSiren.Frequency2.GrnStkLgh := FALSE;
   Std.LightSiren.Frequency2.WhtStkLgh := FALSE;
   Std.LightSiren.Frequency2.Cust1_StaPbtLgh := FALSE;
   Std.LightSiren.Frequency2.Cust1_RstPbtLgh := FALSE;
   Std.LightSiren.Frequency2.Cust1_Siren := FALSE;
   Std.LightSiren.Frequency2.Cust1_RedStkLgh := FALSE;
   Std.LightSiren.Frequency2.Cust1_OngStkLgh := FALSE;
   Std.LightSiren.Frequency2.Cust1_GrnStkLgh := FALSE;
   Std.LightSiren.Frequency2.Cust1_BluStkLgh := FALSE;
   Std.LightSiren.Frequency2.Cust1_WhtStkLgh := FALSE;
   Std.LightSiren.Frequency3.StaPbtLgh := FALSE;
   Std.LightSiren.Frequency3.RstPbtLgh := FALSE;
   Std.LightSiren.Frequency3.EnaPbtLgh := FALSE;
   Std.LightSiren.Frequency3.Siren := FALSE;
   Std.LightSiren.Frequency3.YelStkLgh := FALSE;
   Std.LightSiren.Frequency3.BluStkLgh := FALSE;
   Std.LightSiren.Frequency3.GrnStkLgh := FALSE;
   Std.LightSiren.Frequency3.WhtStkLgh := FALSE;
   Std.LightSiren.Frequency3.Cust1_StaPbtLgh := FALSE;
   Std.LightSiren.Frequency3.Cust1_RstPbtLgh := FALSE;
   Std.LightSiren.Frequency3.Cust1_Siren := FALSE;
   Std.LightSiren.Frequency3.Cust1_RedStkLgh := FALSE;
   Std.LightSiren.Frequency3.Cust1_OngStkLgh := FALSE;
   Std.LightSiren.Frequency3.Cust1_GrnStkLgh := FALSE;
   Std.LightSiren.Frequency3.Cust1_BluStkLgh := FALSE;
   Std.LightSiren.Frequency3.Cust1_WhtStkLgh := FALSE;
   Std.LightSiren.Frequency4.StaPbtLgh := FALSE;
   Std.LightSiren.Frequency4.RstPbtLgh := FALSE;
   Std.LightSiren.Frequency4.EnaPbtLgh := FALSE;
   Std.LightSiren.Frequency4.Siren := FALSE;
   Std.LightSiren.Frequency4.YelStkLgh := FALSE;
   Std.LightSiren.Frequency4.BluStkLgh := FALSE;
   Std.LightSiren.Frequency4.GrnStkLgh := FALSE;
   Std.LightSiren.Frequency4.WhtStkLgh := FALSE;
   Std.LightSiren.Frequency4.Cust1_StaPbtLgh := FALSE;
   Std.LightSiren.Frequency4.Cust1_RstPbtLgh := FALSE;
   Std.LightSiren.Frequency4.Cust1_Siren := FALSE;
   Std.LightSiren.Frequency4.Cust1_RedStkLgh := FALSE;
   Std.LightSiren.Frequency4.Cust1_OngStkLgh := FALSE;
   Std.LightSiren.Frequency4.Cust1_GrnStkLgh := FALSE;
   Std.LightSiren.Frequency4.Cust1_BluStkLgh := FALSE;
   Std.LightSiren.Frequency4.Cust1_WhtStkLgh := FALSE;
   Std.MachineStateModel.EnableIn := FALSE;
   Std.MachineStateModel.EnableOut := FALSE;
   Std.MachineStateModel.Cmd_Mode := 1;
   Std.MachineStateModel.Cmd_Reset := FALSE;
   Std.MachineStateModel.Cmd_Start := FALSE;
   Std.MachineStateModel.Cmd_Stop := FALSE;
   Std.MachineStateModel.Cmd_Hold := FALSE;
   Std.MachineStateModel.Cmd_UnHold := FALSE;
   Std.MachineStateModel.Cmd_Suspend := FALSE;
   Std.MachineStateModel.Cmd_UnSuspend := FALSE;
   Std.MachineStateModel.Cmd_Abort := FALSE;
   Std.MachineStateModel.Cmd_Clear := FALSE;
   Std.MachineStateModel.Cmd_StateComplete := FALSE;
   Std.MachineStateModel.Cmd_ModeManual := FALSE;
   Std.MachineStateModel.Cmd_ModeProduce := TRUE;
   Std.MachineStateModel.Cfg_RemoteCmdEnable := FALSE;
   Std.MachineStateModel.Inp_RemoteModeCmd := 0;
   Std.MachineStateModel.Inp_RemoteModeCmdChangeRequest := FALSE;
   Std.MachineStateModel.Inp_RemoteStateCmd := 0;
   Std.MachineStateModel.Inp_RemoteStateCmdChangeRequest := FALSE;
   Std.MachineStateModel.StartRequest := FALSE;
   Std.MachineStateModel.ResetRequest := FALSE;
   Std.MachineStateModel.Sts_StateCurrent := 9;
   Std.MachineStateModel.Sts_ModeCurrent := 1;
   Std.MachineStateModel.Sts_DisabledStates := 203776;
   Std.MachineStateModel.Sts_ProductionModeCurrent := TRUE;
   Std.MachineStateModel.Sts_ManualModeCurrent := FALSE;
   Std.MachineStateModel.Sts_ClearingEnabled := TRUE;
   Std.MachineStateModel.Sts_StoppedEnabled := TRUE;
   Std.MachineStateModel.Sts_StartingEnabled := TRUE;
   Std.MachineStateModel.Sts_IdleEnabled := TRUE;
   Std.MachineStateModel.Sts_SuspendedEnabled := TRUE;
   Std.MachineStateModel.Sts_ExecuteEnabled := TRUE;
   Std.MachineStateModel.Sts_StoppingEnabled := TRUE;
   Std.MachineStateModel.Sts_AbortingEnabled := TRUE;
   Std.MachineStateModel.Sts_AbortedEnabled := TRUE;
   Std.MachineStateModel.Sts_HoldingEnabled := FALSE;
   Std.MachineStateModel.Sts_HeldEnabled := FALSE;
   Std.MachineStateModel.Sts_UnHoldingEnabled := FALSE;
   Std.MachineStateModel.Sts_SuspendingEnabled := TRUE;
   Std.MachineStateModel.Sts_UnSuspendingEnabled := TRUE;
   Std.MachineStateModel.Sts_ResettingEnabled := TRUE;
   Std.MachineStateModel.Sts_CompletingEnabled := FALSE;
   Std.MachineStateModel.Sts_CompleteEnabled := FALSE;
   Std.MachineStateModel.Sts_ModeChangeNotAllowed := FALSE;
   Std.MachineStateModel.Sts_Clearing := FALSE;
   Std.MachineStateModel.Sts_Stopped := FALSE;
   Std.MachineStateModel.Sts_Starting := FALSE;
   Std.MachineStateModel.Sts_Idle := FALSE;
   Std.MachineStateModel.Sts_Suspended := FALSE;
   Std.MachineStateModel.Sts_Execute := FALSE;
   Std.MachineStateModel.Sts_Stopping := FALSE;
   Std.MachineStateModel.Sts_Aborting := FALSE;
   Std.MachineStateModel.Sts_Aborted := TRUE;
   Std.MachineStateModel.Sts_Holding := FALSE;
   Std.MachineStateModel.Sts_Held := FALSE;
   Std.MachineStateModel.Sts_UnHolding := FALSE;
   Std.MachineStateModel.Sts_Suspending := FALSE;
   Std.MachineStateModel.Sts_UnSuspending := FALSE;
   Std.MachineStateModel.Sts_Resetting := FALSE;
   Std.MachineStateModel.Sts_Complete := FALSE;
   Std.MachineStateModel.Sts_Completing := FALSE;
   Std.MachineStateModel.Sts_AbortingDone := FALSE;
   Std.MachineStateModel.Sts_ClearingDone := FALSE;
   Std.MachineStateModel.Sts_ResettingDone := FALSE;
   Std.MachineStateModel.Sts_StartingDone := FALSE;
   Std.MachineStateModel.Sts_UnSuspendingDone := FALSE;
   Std.MachineStateModel.Sts_StoppingDone := FALSE;
   Std.MachineStateModel.Sts_SuspendingDone := FALSE;
   Std.MachineStateModel.TON_TimeoutStop.PT := T#0MS;
   Std.MachineStateModel.TON_TimeoutStop.IN := FALSE;
   Std.MachineStateModel.TON_TimeoutAbort.PT := T#0MS;
   Std.MachineStateModel.TON_TimeoutAbort.IN := FALSE;
   Std.MachineStateModel.TON_Start.PT := T#0MS;
   Std.MachineStateModel.TON_Start.IN := FALSE;
   Std.TON_SafetyOn.PT := T#1S;
   Std.TON_SafetyOn.ET := T#1S;
   Std.TON_SafetyOn.IN := TRUE;
   Std.TON_SafetyOn.Q := TRUE;
   Std.TOF_SirenEna.PT := T#5S;
   Std.TOF_SirenEna.ET := T#5S;
   Std.TOF_SirenEna.IN := FALSE;
   Gen.Cfg_1Jog_0Move := FALSE;
   Gen.DeadManAct := FALSE;
   Gen.AlmOk := TRUE;
   Gen.MotionScOk := FALSE;
   Gen.MotionOkToStop := TRUE;
   Gen.ScSeqOk := FALSE;
   Gen.CycleOn := FALSE;
   Gen.StopInPhase := FALSE;
   Gen.OutChainObstruction := TRUE;
   Gen.SummAlmImmStopChainOK := TRUE;
   Gen.SummLongChainEndMouldPres := TRUE;
   Gen.SummCrossChainEndMouldPres := TRUE;
   Gen.SummEnaMoveChain := TRUE;
   Gen.PosOkLongChain := FALSE;
   Gen.PosOkCrossChain := TRUE;
   Gen.StationWorkedOnLongChain := TRUE;
   Gen.StationWorkedOnCrossChain := TRUE;
   Gen.CammingStart := FALSE;
   Gen.CamHookAxis := FALSE;
   Gen.DrivesEnabled := FALSE;
   Gen.LongChainRange := TRUE;
   Gen.CrossChainRange := FALSE;
   Gen.CheckStationsOutOfObstruction := FALSE;
   Gen.CheckConditionLongChainStep := FALSE;
   Gen.CheckConditionCrossChainStep := FALSE;
   Gen.SlowFirstStepAfterEmerg := TRUE;
   Gen.Work := FALSE;
   Gen.AuxStartCamRequest := FALSE;
   Gen.StrobeSpeedUp := FALSE;
   Gen.StrobeMould := FALSE;
   Gen.StrobeShift := FALSE;
   Gen.ManConsoleSelection := 0;
   Gen.KConv_DegSec := 6.0;
   Gen.LastSpeedLineUsed := 0.0;
   Gen.Cfg_GearRatio := 1.0;
   Gen.Chian8Cross_StartPos := 0.0;
   Gen.Chian8Cross_EndPos := 0.0;
   Gen.TON_ScOK.PT := T#20S;
   Gen.TON_ScOK.IN := FALSE;
   Param.Gen_Ena_LongCycle := TRUE;
   Param.Gen_Ena_RejByTimeout_Zone1 := FALSE;
   Param.Gen_Ena_RejByTimeout_Zone2 := FALSE;
   Param.Gen_Ena_RejByTimeout_Zone3 := FALSE;
   Param.Gen_Ena_RejByTimeout_Zone4 := FALSE;
   Param.Gen_RejByTimeout_Zone1 := 0;
   Param.Gen_RejByTimeout_Zone2 := 0;
   Param.Gen_RejByTimeout_Zone3 := 0;
   Param.Gen_RejByTimeout_Zone4 := 0;
   Param.Gen_ProdPerMould := 0;
   Param.Gen_Speed_Line := 10.0;
   Param.Gen_Kpos_MasterLongRange := 0.45;
   Param.Chain1Long_Torque_Limit := 30.0;
   Param.Chain2Long_Torque_Limit := 30.0;
   Param.Chain3Long_Torque_Limit := 30.0;
   Param.Chain4Cross_Torque_Limit := 30.0;
   Param.Chain5Long_Torque_Limit := 30.0;
   Param.Chain6Long_Torque_Limit := 30.0;
   Param.Chain7Long_Torque_Limit := 30.0;
   Param.Chain8Cross_Torque_Limit := 30.0;
   LastHmiDataParam.Gen_Ena_LongCycle := FALSE;
   LastHmiDataParam.Gen_Ena_RejByTimeout_Zone1 := FALSE;
   LastHmiDataParam.Gen_Ena_RejByTimeout_Zone2 := FALSE;
   LastHmiDataParam.Gen_Ena_RejByTimeout_Zone3 := FALSE;
   LastHmiDataParam.Gen_Ena_RejByTimeout_Zone4 := FALSE;
   LastHmiDataParam.Gen_RejByTimeout_Zone1 := 0;
   LastHmiDataParam.Gen_RejByTimeout_Zone2 := 0;
   LastHmiDataParam.Gen_RejByTimeout_Zone3 := 0;
   LastHmiDataParam.Gen_RejByTimeout_Zone4 := 0;
   LastHmiDataParam.Gen_ProdPerMould := 0;
   LastHmiDataParam.Gen_Speed_Line := 0.0;
   LastHmiDataParam.Gen_Kpos_MasterLongRange := 0.0;
   LastHmiDataParam.Chain1Long_Torque_Limit := 0.0;
   LastHmiDataParam.Chain2Long_Torque_Limit := 0.0;
   LastHmiDataParam.Chain3Long_Torque_Limit := 0.0;
   LastHmiDataParam.Chain4Cross_Torque_Limit := 0.0;
   LastHmiDataParam.Chain5Long_Torque_Limit := 0.0;
   LastHmiDataParam.Chain6Long_Torque_Limit := 0.0;
   LastHmiDataParam.Chain7Long_Torque_Limit := 0.0;
   LastHmiDataParam.Chain8Cross_Torque_Limit := 0.0;
   Alm.ThSwitch."0" := FALSE;   // CH1.Alm.ThSwitch.0
   Alm.ThSwitch."1" := FALSE;   // CH1.Alm.ThSwitch.1
   Alm.ThSwitch."2" := FALSE;   // CH1.Alm.ThSwitch.2
   Alm.ThSwitch."3" := FALSE;   // CH1.Alm.ThSwitch.3
   Alm.ThSwitch."4" := FALSE;   // CH1.Alm.ThSwitch.4
   Alm.ThSwitch."5" := FALSE;   // CH1.Alm.ThSwitch.5
   Alm.ThSwitch."6" := FALSE;   // CH1.Alm.ThSwitch.6
   Alm.ThSwitch."7" := FALSE;   // CH1.Alm.ThSwitch.7
   Alm.ThSwitch."8" := FALSE;   // CH1.Alm.ThSwitch.8
   Alm.ThSwitch."9" := FALSE;   // CH1.Alm.ThSwitch.9
   Alm.ThSwitch."10" := FALSE;   // CH1.Alm.ThSwitch.10
   Alm.ThSwitch."11" := FALSE;   // CH1.Alm.ThSwitch.11
   Alm.ThSwitch."12" := FALSE;   // CH1.Alm.ThSwitch.12
   Alm.ThSwitch."13" := FALSE;   // CH1.Alm.ThSwitch.13
   Alm.ThSwitch."14" := FALSE;   // CH1.Alm.ThSwitch.14
   Alm.ThSwitch."15" := FALSE;   // CH1.Alm.ThSwitch.15
   Alm.ThSwitch."16" := FALSE;   // CH1.Alm.ThSwitch.16
   Alm.ThSwitch."17" := FALSE;   // CH1.Alm.ThSwitch.17
   Alm.ThSwitch."18" := FALSE;   // CH1.Alm.ThSwitch.18
   Alm.ThSwitch."19" := FALSE;   // CH1.Alm.ThSwitch.19
   Alm.ThSwitch."20" := FALSE;   // CH1.Alm.ThSwitch.20
   Alm.ThSwitch."21" := FALSE;   // CH1.Alm.ThSwitch.21
   Alm.ThSwitch."22" := FALSE;   // CH1.Alm.ThSwitch.22
   Alm.ThSwitch."23" := FALSE;   // CH1.Alm.ThSwitch.23
   Alm.ThSwitch."24" := FALSE;   // CH1.Alm.ThSwitch.24
   Alm.ThSwitch."25" := FALSE;   // CH1.Alm.ThSwitch.25
   Alm.ThSwitch."26" := FALSE;   // CH1.Alm.ThSwitch.26
   Alm.ThSwitch."27" := FALSE;   // CH1.Alm.ThSwitch.27
   Alm.ThSwitch."28" := FALSE;   // CH1.Alm.ThSwitch.28
   Alm.ThSwitch."29" := FALSE;   // CH1.Alm.ThSwitch.29
   Alm.ThSwitch."30" := FALSE;   // CH1.Alm.ThSwitch.30
   Alm.ThSwitch."31" := FALSE;   // CH1.Alm.ThSwitch.31
   Alm.SafeComm."0" := FALSE;   // CH1.Alm.SafeComm.0 > Communication fault sinamics chain 1 (1CH40TB5)
   Alm.SafeComm."1" := FALSE;   // CH1.Alm.SafeComm.1 > Communication fault sinamics chain 2 (1CH40TB5)
   Alm.SafeComm."2" := FALSE;   // CH1.Alm.SafeComm.2 > Communication fault sinamics chain 3 (1CH42TB5)
   Alm.SafeComm."3" := FALSE;   // CH1.Alm.SafeComm.3 > Communication fault sinamics chain 4 (1CH44TB5)
   Alm.SafeComm."4" := FALSE;   // CH1.Alm.SafeComm.4 > Communication fault sinamics chain 5 (1CH48TB5)
   Alm.SafeComm."5" := FALSE;   // CH1.Alm.SafeComm.5 > Communication fault sinamics chain 6 (1CH46TB5)
   Alm.SafeComm."6" := FALSE;   // CH1.Alm.SafeComm.6 > Communication fault sinamics chain 7 (1CH48TB5)
   Alm.SafeComm."7" := FALSE;   // CH1.Alm.SafeComm.7 > Communication fault sinamics chain 8 (1CH44TB5)
   Alm.SafeComm."8" := FALSE;   // CH1.Alm.SafeComm.8
   Alm.SafeComm."9" := FALSE;   // CH1.Alm.SafeComm.9
   Alm.SafeComm."10" := FALSE;   // CH1.Alm.SafeComm.10
   Alm.SafeComm."11" := FALSE;   // CH1.Alm.SafeComm.11
   Alm.SafeComm."12" := FALSE;   // CH1.Alm.SafeComm.12
   Alm.SafeComm."13" := FALSE;   // CH1.Alm.SafeComm.13
   Alm.SafeComm."14" := FALSE;   // CH1.Alm.SafeComm.14
   Alm.SafeComm."15" := FALSE;   // CH1.Alm.SafeComm.15
   Alm.SafeComm."16" := FALSE;   // CH1.Alm.SafeComm.16
   Alm.SafeComm."17" := FALSE;   // CH1.Alm.SafeComm.17
   Alm.SafeComm."18" := FALSE;   // CH1.Alm.SafeComm.18
   Alm.SafeComm."19" := FALSE;   // CH1.Alm.SafeComm.19
   Alm.SafeComm."20" := FALSE;   // CH1.Alm.SafeComm.20
   Alm.SafeComm."21" := FALSE;   // CH1.Alm.SafeComm.21
   Alm.SafeComm."22" := FALSE;   // CH1.Alm.SafeComm.22
   Alm.SafeComm."23" := FALSE;   // CH1.Alm.SafeComm.23
   Alm.SafeComm."24" := FALSE;   // CH1.Alm.SafeComm.24
   Alm.SafeComm."25" := FALSE;   // CH1.Alm.SafeComm.25
   Alm.SafeComm."26" := FALSE;   // CH1.Alm.SafeComm.26
   Alm.SafeComm."27" := FALSE;   // CH1.Alm.SafeComm.27
   Alm.SafeComm."28" := FALSE;   // CH1.Alm.SafeComm.28
   Alm.SafeComm."29" := FALSE;   // CH1.Alm.SafeComm.29
   Alm.SafeComm."30" := FALSE;   // CH1.Alm.SafeComm.30
   Alm.SafeComm."31" := FALSE;   // CH1.Alm.SafeComm.31
   Alm.SafeEmg."0" := FALSE;   // CH1.Alm.SafeEmg.0
   Alm.SafeEmg."1" := FALSE;   // CH1.Alm.SafeEmg.1
   Alm.SafeEmg."2" := FALSE;   // CH1.Alm.SafeEmg.2
   Alm.SafeEmg."3" := FALSE;   // CH1.Alm.SafeEmg.3
   Alm.SafeEmg."4" := FALSE;   // CH1.Alm.SafeEmg.4
   Alm.SafeEmg."5" := FALSE;   // CH1.Alm.SafeEmg.5
   Alm.SafeEmg."6" := FALSE;   // CH1.Alm.SafeEmg.6
   Alm.SafeEmg."7" := FALSE;   // CH1.Alm.SafeEmg.7
   Alm.SafeEmg."8" := FALSE;   // CH1.Alm.SafeEmg.8
   Alm.SafeEmg."9" := FALSE;   // CH1.Alm.SafeEmg.9
   Alm.SafeEmg."10" := FALSE;   // CH1.Alm.SafeEmg.10
   Alm.SafeEmg."11" := FALSE;   // CH1.Alm.SafeEmg.11
   Alm.SafeEmg."12" := FALSE;   // CH1.Alm.SafeEmg.12
   Alm.SafeEmg."13" := FALSE;   // CH1.Alm.SafeEmg.13
   Alm.SafeEmg."14" := FALSE;   // CH1.Alm.SafeEmg.14
   Alm.SafeEmg."15" := FALSE;   // CH1.Alm.SafeEmg.15
   Alm.SafeEmg."16" := FALSE;   // CH1.Alm.SafeEmg.16
   Alm.SafeEmg."17" := FALSE;   // CH1.Alm.SafeEmg.17
   Alm.SafeEmg."18" := FALSE;   // CH1.Alm.SafeEmg.18
   Alm.SafeEmg."19" := FALSE;   // CH1.Alm.SafeEmg.19
   Alm.SafeEmg."20" := FALSE;   // CH1.Alm.SafeEmg.20
   Alm.SafeEmg."21" := FALSE;   // CH1.Alm.SafeEmg.21
   Alm.SafeEmg."22" := FALSE;   // CH1.Alm.SafeEmg.22
   Alm.SafeEmg."23" := FALSE;   // CH1.Alm.SafeEmg.23
   Alm.SafeEmg."24" := FALSE;   // CH1.Alm.SafeEmg.24
   Alm.SafeEmg."25" := FALSE;   // CH1.Alm.SafeEmg.25
   Alm.SafeEmg."26" := FALSE;   // CH1.Alm.SafeEmg.26
   Alm.SafeEmg."27" := FALSE;   // CH1.Alm.SafeEmg.27
   Alm.SafeEmg."28" := FALSE;   // CH1.Alm.SafeEmg.28
   Alm.SafeEmg."29" := FALSE;   // CH1.Alm.SafeEmg.29
   Alm.SafeEmg."30" := FALSE;   // CH1.Alm.SafeEmg.30
   Alm.SafeEmg."31" := FALSE;   // CH1.Alm.SafeEmg.31
   Alm.SafeGuards."0" := FALSE;   // CH1.Alm.SafeGuards.0 > Drive chain 1 long (1CH40MA8)
   Alm.SafeGuards."1" := FALSE;   // CH1.Alm.SafeGuards.1 > Drive chain 2 long (1CH41MA8)
   Alm.SafeGuards."2" := FALSE;   // CH1.Alm.SafeGuards.2 > Drive chain 3 long (1CH42MA8)
   Alm.SafeGuards."3" := FALSE;   // CH1.Alm.SafeGuards.3 > Drive chain 4 cross (1CH44MA8)
   Alm.SafeGuards."4" := FALSE;   // CH1.Alm.SafeGuards.4 > Drive chain 5 long (1CH48MA8)
   Alm.SafeGuards."5" := FALSE;   // CH1.Alm.SafeGuards.5 > Drive chain 6 long (1CH46MA8)
   Alm.SafeGuards."6" := FALSE;   // CH1.Alm.SafeGuards.6 > Drive chain 7 long (1CH49MA8)
   Alm.SafeGuards."7" := FALSE;   // CH1.Alm.SafeGuards.7 > Drive chain 8 cross (1CH45MA8)
   Alm.SafeGuards."8" := FALSE;   // CH1.Alm.SafeGuards.8
   Alm.SafeGuards."9" := FALSE;   // CH1.Alm.SafeGuards.9
   Alm.SafeGuards."10" := FALSE;   // CH1.Alm.SafeGuards.10
   Alm.SafeGuards."11" := FALSE;   // CH1.Alm.SafeGuards.11
   Alm.SafeGuards."12" := FALSE;   // CH1.Alm.SafeGuards.12
   Alm.SafeGuards."13" := FALSE;   // CH1.Alm.SafeGuards.13
   Alm.SafeGuards."14" := FALSE;   // CH1.Alm.SafeGuards.14
   Alm.SafeGuards."15" := FALSE;   // CH1.Alm.SafeGuards.15
   Alm.SafeGuards."16" := FALSE;   // CH1.Alm.SafeGuards.16
   Alm.SafeGuards."17" := FALSE;   // CH1.Alm.SafeGuards.17
   Alm.SafeGuards."18" := FALSE;   // CH1.Alm.SafeGuards.18
   Alm.SafeGuards."19" := FALSE;   // CH1.Alm.SafeGuards.19
   Alm.SafeGuards."20" := FALSE;   // CH1.Alm.SafeGuards.20
   Alm.SafeGuards."21" := FALSE;   // CH1.Alm.SafeGuards.21
   Alm.SafeGuards."22" := FALSE;   // CH1.Alm.SafeGuards.22
   Alm.SafeGuards."23" := FALSE;   // CH1.Alm.SafeGuards.23
   Alm.SafeGuards."24" := FALSE;   // CH1.Alm.SafeGuards.24
   Alm.SafeGuards."25" := FALSE;   // CH1.Alm.SafeGuards.25
   Alm.SafeGuards."26" := FALSE;   // CH1.Alm.SafeGuards.26
   Alm.SafeGuards."27" := FALSE;   // CH1.Alm.SafeGuards.27
   Alm.SafeGuards."28" := FALSE;   // CH1.Alm.SafeGuards.28
   Alm.SafeGuards."29" := FALSE;   // CH1.Alm.SafeGuards.29
   Alm.SafeGuards."30" := FALSE;   // CH1.Alm.SafeGuards.30
   Alm.SafeGuards."31" := FALSE;   // CH1.Alm.SafeGuards.31
   Alm.GtaAirGroup."0" := FALSE;   // CH1.Alm.GtaAirGroup.0
   Alm.GtaAirGroup."1" := FALSE;   // CH1.Alm.GtaAirGroup.1
   Alm.GtaAirGroup."2" := FALSE;   // CH1.Alm.GtaAirGroup.2
   Alm.GtaAirGroup."3" := FALSE;   // CH1.Alm.GtaAirGroup.3
   Alm.GtaAirGroup."4" := FALSE;   // CH1.Alm.GtaAirGroup.4
   Alm.GtaAirGroup."5" := FALSE;   // CH1.Alm.GtaAirGroup.5
   Alm.GtaAirGroup."6" := FALSE;   // CH1.Alm.GtaAirGroup.6
   Alm.GtaAirGroup."7" := FALSE;   // CH1.Alm.GtaAirGroup.7
   Alm.GtaAirGroup."8" := FALSE;   // CH1.Alm.GtaAirGroup.8
   Alm.GtaAirGroup."9" := FALSE;   // CH1.Alm.GtaAirGroup.9
   Alm.GtaAirGroup."10" := FALSE;   // CH1.Alm.GtaAirGroup.10
   Alm.GtaAirGroup."11" := FALSE;   // CH1.Alm.GtaAirGroup.11
   Alm.GtaAirGroup."12" := FALSE;   // CH1.Alm.GtaAirGroup.12
   Alm.GtaAirGroup."13" := FALSE;   // CH1.Alm.GtaAirGroup.13
   Alm.GtaAirGroup."14" := FALSE;   // CH1.Alm.GtaAirGroup.14
   Alm.GtaAirGroup."15" := FALSE;   // CH1.Alm.GtaAirGroup.15
   Alm.GtaAirGroup."16" := FALSE;   // CH1.Alm.GtaAirGroup.16
   Alm.GtaAirGroup."17" := FALSE;   // CH1.Alm.GtaAirGroup.17
   Alm.GtaAirGroup."18" := FALSE;   // CH1.Alm.GtaAirGroup.18
   Alm.GtaAirGroup."19" := FALSE;   // CH1.Alm.GtaAirGroup.19
   Alm.GtaAirGroup."20" := FALSE;   // CH1.Alm.GtaAirGroup.20
   Alm.GtaAirGroup."21" := FALSE;   // CH1.Alm.GtaAirGroup.21
   Alm.GtaAirGroup."22" := FALSE;   // CH1.Alm.GtaAirGroup.22
   Alm.GtaAirGroup."23" := FALSE;   // CH1.Alm.GtaAirGroup.23
   Alm.GtaAirGroup."24" := FALSE;   // CH1.Alm.GtaAirGroup.24
   Alm.GtaAirGroup."25" := FALSE;   // CH1.Alm.GtaAirGroup.25
   Alm.GtaAirGroup."26" := FALSE;   // CH1.Alm.GtaAirGroup.26
   Alm.GtaAirGroup."27" := FALSE;   // CH1.Alm.GtaAirGroup.27
   Alm.GtaAirGroup."28" := FALSE;   // CH1.Alm.GtaAirGroup.28
   Alm.GtaAirGroup."29" := FALSE;   // CH1.Alm.GtaAirGroup.29
   Alm.GtaAirGroup."30" := FALSE;   // CH1.Alm.GtaAirGroup.30
   Alm.GtaAirGroup."31" := FALSE;   // CH1.Alm.GtaAirGroup.31
   Alm.Major."0" := FALSE;   // CH1.Alm.Major.0
   Alm.Major."1" := FALSE;   // CH1.Alm.Major.1
   Alm.Major."2" := FALSE;   // CH1.Alm.Major.2
   Alm.Major."3" := FALSE;   // CH1.Alm.Major.3
   Alm.Major."4" := FALSE;   // CH1.Alm.Major.4
   Alm.Major."5" := FALSE;   // CH1.Alm.Major.5
   Alm.Major."6" := FALSE;   // CH1.Alm.Major.6
   Alm.Major."7" := FALSE;   // CH1.Alm.Major.7
   Alm.Major."8" := FALSE;   // CH1.Alm.Major.8
   Alm.Major."9" := FALSE;   // CH1.Alm.Major.9
   Alm.Major."10" := FALSE;   // CH1.Alm.Major.10
   Alm.Major."11" := FALSE;   // CH1.Alm.Major.11
   Alm.Major."12" := FALSE;   // CH1.Alm.Major.12
   Alm.Major."13" := FALSE;   // CH1.Alm.Major.13
   Alm.Major."14" := FALSE;   // CH1.Alm.Major.14
   Alm.Major."15" := FALSE;   // CH1.Alm.Major.15
   Alm.Major."16" := FALSE;   // CH1.Alm.Major.16
   Alm.Major."17" := FALSE;   // CH1.Alm.Major.17
   Alm.Major."18" := FALSE;   // CH1.Alm.Major.18
   Alm.Major."19" := FALSE;   // CH1.Alm.Major.19
   Alm.Major."20" := FALSE;   // CH1.Alm.Major.20
   Alm.Major."21" := FALSE;   // CH1.Alm.Major.21
   Alm.Major."22" := FALSE;   // CH1.Alm.Major.22
   Alm.Major."23" := FALSE;   // CH1.Alm.Major.23
   Alm.Major."24" := FALSE;   // CH1.Alm.Major.24
   Alm.Major."25" := FALSE;   // CH1.Alm.Major.25
   Alm.Major."26" := FALSE;   // CH1.Alm.Major.26
   Alm.Major."27" := FALSE;   // CH1.Alm.Major.27
   Alm.Major."28" := FALSE;   // CH1.Alm.Major.28
   Alm.Major."29" := FALSE;   // CH1.Alm.Major.29
   Alm.Major."30" := FALSE;   // CH1.Alm.Major.30
   Alm.Major."31" := FALSE;   // CH1.Alm.Major.31
   Alm.Minor."0" := FALSE;   // CH1.Alm.Minor.0 > Station in manual mode selected
   Alm.Minor."1" := FALSE;   // CH1.Alm.Minor.1
   Alm.Minor."2" := FALSE;   // CH1.Alm.Minor.2
   Alm.Minor."3" := FALSE;   // CH1.Alm.Minor.3
   Alm.Minor."4" := FALSE;   // CH1.Alm.Minor.4
   Alm.Minor."5" := FALSE;   // CH1.Alm.Minor.5
   Alm.Minor."6" := FALSE;   // CH1.Alm.Minor.6
   Alm.Minor."7" := FALSE;   // CH1.Alm.Minor.7
   Alm.Minor."8" := FALSE;   // CH1.Alm.Minor.8
   Alm.Minor."9" := FALSE;   // CH1.Alm.Minor.9
   Alm.Minor."10" := FALSE;   // CH1.Alm.Minor.10
   Alm.Minor."11" := FALSE;   // CH1.Alm.Minor.11 > Timeout start condition
   Alm.Minor."12" := FALSE;   // CH1.Alm.Minor.12
   Alm.Minor."13" := FALSE;   // CH1.Alm.Minor.13
   Alm.Minor."14" := FALSE;   // CH1.Alm.Minor.14
   Alm.Minor."15" := FALSE;   // CH1.Alm.Minor.15
   Alm.Minor."16" := FALSE;   // CH1.Alm.Minor.16
   Alm.Minor."17" := FALSE;   // CH1.Alm.Minor.17
   Alm.Minor."18" := FALSE;   // CH1.Alm.Minor.18
   Alm.Minor."19" := FALSE;   // CH1.Alm.Minor.19
   Alm.Minor."20" := FALSE;   // CH1.Alm.Minor.20
   Alm.Minor."21" := FALSE;   // CH1.Alm.Minor.21
   Alm.Minor."22" := FALSE;   // CH1.Alm.Minor.22
   Alm.Minor."23" := FALSE;   // CH1.Alm.Minor.23
   Alm.Minor."24" := FALSE;   // CH1.Alm.Minor.24
   Alm.Minor."25" := FALSE;   // CH1.Alm.Minor.25
   Alm.Minor."26" := FALSE;   // CH1.Alm.Minor.26
   Alm.Minor."27" := FALSE;   // CH1.Alm.Minor.27
   Alm.Minor."28" := FALSE;   // CH1.Alm.Minor.28
   Alm.Minor."29" := FALSE;   // CH1.Alm.Minor.29
   Alm.Minor."30" := FALSE;   // CH1.Alm.Minor.30
   Alm.Minor."31" := FALSE;   // CH1.Alm.Minor.31
   Alm.MinorFtcEndChain."0" := FALSE;   // CH1.Alm.MinorFtcEndChain.0
   Alm.MinorFtcEndChain."1" := FALSE;   // CH1.Alm.MinorFtcEndChain.1 > End chain 1 sensor fault (1AC330BR8)
   Alm.MinorFtcEndChain."2" := FALSE;   // CH1.Alm.MinorFtcEndChain.2 > End chain 2 sensor fault (1FS332BR5)
   Alm.MinorFtcEndChain."3" := FALSE;   // CH1.Alm.MinorFtcEndChain.3 > End chain 3 sensor fault (3VV330BR2)
   Alm.MinorFtcEndChain."4" := FALSE;   // CH1.Alm.MinorFtcEndChain.4 > End chain 4 sensor fault (4VV330BR2)
   Alm.MinorFtcEndChain."5" := FALSE;   // CH1.Alm.MinorFtcEndChain.5 > End chain 5 sensor fault (4AC330BR2)
   Alm.MinorFtcEndChain."6" := FALSE;   // CH1.Alm.MinorFtcEndChain.6 > End chain 6 sensor fault (1OM332BR3)
   Alm.MinorFtcEndChain."7" := FALSE;   // CH1.Alm.MinorFtcEndChain.7 > End chain 7 sensor fault (1RD330BR3)
   Alm.MinorFtcEndChain."8" := FALSE;   // CH1.Alm.MinorFtcEndChain.8 > End chain 8 sensor fault (1FM330BR2)
   Alm.MinorFtcEndChain."9" := FALSE;   // CH1.Alm.MinorFtcEndChain.9
   Alm.MinorFtcEndChain."10" := FALSE;   // CH1.Alm.MinorFtcEndChain.10
   Alm.MinorFtcEndChain."11" := FALSE;   // CH1.Alm.MinorFtcEndChain.11
   Alm.MinorFtcEndChain."12" := FALSE;   // CH1.Alm.MinorFtcEndChain.12
   Alm.MinorFtcEndChain."13" := FALSE;   // CH1.Alm.MinorFtcEndChain.13
   Alm.MinorFtcEndChain."14" := FALSE;   // CH1.Alm.MinorFtcEndChain.14
   Alm.MinorFtcEndChain."15" := FALSE;   // CH1.Alm.MinorFtcEndChain.15
   Alm.MinorFtcEndChain."16" := FALSE;   // CH1.Alm.MinorFtcEndChain.16
   Alm.MinorFtcEndChain."17" := FALSE;   // CH1.Alm.MinorFtcEndChain.17
   Alm.MinorFtcEndChain."18" := FALSE;   // CH1.Alm.MinorFtcEndChain.18
   Alm.MinorFtcEndChain."19" := FALSE;   // CH1.Alm.MinorFtcEndChain.19
   Alm.MinorFtcEndChain."20" := FALSE;   // CH1.Alm.MinorFtcEndChain.20
   Alm.MinorFtcEndChain."21" := FALSE;   // CH1.Alm.MinorFtcEndChain.21
   Alm.MinorFtcEndChain."22" := FALSE;   // CH1.Alm.MinorFtcEndChain.22
   Alm.MinorFtcEndChain."23" := FALSE;   // CH1.Alm.MinorFtcEndChain.23
   Alm.MinorFtcEndChain."24" := FALSE;   // CH1.Alm.MinorFtcEndChain.24
   Alm.MinorFtcEndChain."25" := FALSE;   // CH1.Alm.MinorFtcEndChain.25
   Alm.MinorFtcEndChain."26" := FALSE;   // CH1.Alm.MinorFtcEndChain.26
   Alm.MinorFtcEndChain."27" := FALSE;   // CH1.Alm.MinorFtcEndChain.27
   Alm.MinorFtcEndChain."28" := FALSE;   // CH1.Alm.MinorFtcEndChain.28
   Alm.MinorFtcEndChain."29" := FALSE;   // CH1.Alm.MinorFtcEndChain.29
   Alm.MinorFtcEndChain."30" := FALSE;   // CH1.Alm.MinorFtcEndChain.30
   Alm.MinorFtcEndChain."31" := FALSE;   // CH1.Alm.MinorFtcEndChain.31
   Alm.MinorFtcPresenceChain."0" := FALSE;   // CH1.Alm.MinorFtcPresenceChain.0 > ME1 infeed mould presence extractor booked mould sensor fault (1ME345BR8)
   Alm.MinorFtcPresenceChain."1" := FALSE;   // CH1.Alm.MinorFtcPresenceChain.1 > ME1 infeed mould presence camera detection sensor fault (1ME334BR2)
   Alm.MinorFtcPresenceChain."2" := FALSE;   // CH1.Alm.MinorFtcPresenceChain.2 > ME1 infeed mould presence inserter sensor fault (1ME337BR2)
   Alm.MinorFtcPresenceChain."3" := FALSE;   // CH1.Alm.MinorFtcPresenceChain.3 > CW1 infeed mould presence checkweigher sensor fault (1ID330BR2)
   Alm.MinorFtcPresenceChain."4" := FALSE;   // CH1.Alm.MinorFtcPresenceChain.4 > ID1 infeed mould presence sensor fault (1ID332BR2)
   Alm.MinorFtcPresenceChain."5" := FALSE;   // CH1.Alm.MinorFtcPresenceChain.5 > DP1 infeed mould presence depositor sensor fault (1DP330BR4)
   Alm.MinorFtcPresenceChain."6" := FALSE;   // CH1.Alm.MinorFtcPresenceChain.6 > FS1 infeed mould presence fast shell sensor fault (1FS332BR2)
   Alm.MinorFtcPresenceChain."7" := FALSE;   // CH1.Alm.MinorFtcPresenceChain.7 > CW2 infeed mould presence checkweigher sensor fault (1FS330BR2)
   Alm.MinorFtcPresenceChain."8" := FALSE;   // CH1.Alm.MinorFtcPresenceChain.8 > ID2 infeed mould presence sensor fault (2ID332BR2)
   Alm.MinorFtcPresenceChain."9" := FALSE;   // CH1.Alm.MinorFtcPresenceChain.9 > DP2 infeed mould presence depositor sensor fault (2DP330BR4)
   Alm.MinorFtcPresenceChain."10" := FALSE;   // CH1.Alm.MinorFtcPresenceChain.10 > ID3 infeed mould presence sensor fault (3ID332BR2)
   Alm.MinorFtcPresenceChain."11" := FALSE;   // CH1.Alm.MinorFtcPresenceChain.11 > DP3 infeed mould presence depositor sensor fault (3DP330BR2)
   Alm.MinorFtcPresenceChain."12" := FALSE;   // CH1.Alm.MinorFtcPresenceChain.12 > ID4 infeed mould presence sensor fault (4ID332BR2)
   Alm.MinorFtcPresenceChain."13" := FALSE;   // CH1.Alm.MinorFtcPresenceChain.13 > CW3 infeed mould presence checkweigher sensor fault (4ID330BR2)
   Alm.MinorFtcPresenceChain."14" := FALSE;   // CH1.Alm.MinorFtcPresenceChain.14 > DP4 infeed mould presence depositor sensor fault (4DP330BR2)
   Alm.MinorFtcPresenceChain."15" := FALSE;   // CH1.Alm.MinorFtcPresenceChain.15 > BF1 infeed mould presence checkweigher sensor fault (1BFxxxBR)
   Alm.MinorFtcPresenceChain."16" := FALSE;   // CH1.Alm.MinorFtcPresenceChain.16 > CW4 infeed mould presence checkweigher sensor fault (1BF330BR2)
   Alm.MinorFtcPresenceChain."17" := FALSE;   // CH1.Alm.MinorFtcPresenceChain.17 > CM1 infeed mould presence booking moulds sensor fault (1CM333BR2)
   Alm.MinorFtcPresenceChain."18" := FALSE;   // CH1.Alm.MinorFtcPresenceChain.18 > OM1 infeed mould presence opening moulds sensor fault (1OM332BR2)
   Alm.MinorFtcPresenceChain."19" := FALSE;   // CH1.Alm.MinorFtcPresenceChain.19 > RD1 twist mould presence demoulder sensor fault (1RD332BR2)
   Alm.MinorFtcPresenceChain."20" := FALSE;   // CH1.Alm.MinorFtcPresenceChain.20
   Alm.MinorFtcPresenceChain."21" := FALSE;   // CH1.Alm.MinorFtcPresenceChain.21
   Alm.MinorFtcPresenceChain."22" := FALSE;   // CH1.Alm.MinorFtcPresenceChain.22
   Alm.MinorFtcPresenceChain."23" := FALSE;   // CH1.Alm.MinorFtcPresenceChain.23
   Alm.MinorFtcPresenceChain."24" := FALSE;   // CH1.Alm.MinorFtcPresenceChain.24
   Alm.MinorFtcPresenceChain."25" := FALSE;   // CH1.Alm.MinorFtcPresenceChain.25
   Alm.MinorFtcPresenceChain."26" := FALSE;   // CH1.Alm.MinorFtcPresenceChain.26
   Alm.MinorFtcPresenceChain."27" := FALSE;   // CH1.Alm.MinorFtcPresenceChain.27
   Alm.MinorFtcPresenceChain."28" := FALSE;   // CH1.Alm.MinorFtcPresenceChain.28
   Alm.MinorFtcPresenceChain."29" := FALSE;   // CH1.Alm.MinorFtcPresenceChain.29
   Alm.MinorFtcPresenceChain."30" := FALSE;   // CH1.Alm.MinorFtcPresenceChain.30
   Alm.MinorFtcPresenceChain."31" := FALSE;   // CH1.Alm.MinorFtcPresenceChain.31
   Alm.MinorFtcMouldOnLug."0" := FALSE;   // CH1.Alm.MinorFtcMouldOnLug.0 > ME1 outfeed inserter mould on lug sensor fault (1ME337BR4)
   Alm.MinorFtcMouldOnLug."1" := FALSE;   // CH1.Alm.MinorFtcMouldOnLug.1 > AC1 infeed mould on lug sensor fault (1AC330BR6)
   Alm.MinorFtcMouldOnLug."2" := FALSE;   // CH1.Alm.MinorFtcMouldOnLug.2 > AC1 outfeed mould on lug sensor fault (1AC330BR7)
   Alm.MinorFtcMouldOnLug."3" := FALSE;   // CH1.Alm.MinorFtcMouldOnLug.3 > SF1 infeed mould on lug sensor fault (1FS332BR3)
   Alm.MinorFtcMouldOnLug."4" := FALSE;   // CH1.Alm.MinorFtcMouldOnLug.4 > SF1 outfeed mould on lug sensor fault (1FS332BR4)
   Alm.MinorFtcMouldOnLug."5" := FALSE;   // CH1.Alm.MinorFtcMouldOnLug.5 > AC2 infeed mould on lug sensor fault (2AC330BR6)
   Alm.MinorFtcMouldOnLug."6" := FALSE;   // CH1.Alm.MinorFtcMouldOnLug.6 > AC2 outfeed mould on lug sensor fault (2AC330BR7)
   Alm.MinorFtcMouldOnLug."7" := FALSE;   // CH1.Alm.MinorFtcMouldOnLug.7 > AC3 infeed mould on lug sensor fault (3AC330BR6)
   Alm.MinorFtcMouldOnLug."8" := FALSE;   // CH1.Alm.MinorFtcMouldOnLug.8 > AC3 outfeed mould on lug sensor fault (3AC430BR6)
   Alm.MinorFtcMouldOnLug."9" := FALSE;   // CH1.Alm.MinorFtcMouldOnLug.9 > CM1 infeed mould on lug sensor fault (1CM334BR2)
   Alm.MinorFtcMouldOnLug."10" := FALSE;   // CH1.Alm.MinorFtcMouldOnLug.10 > CM1 infeed buffer mould on lug sensor fault (1CM335BR8)
   Alm.MinorFtcMouldOnLug."11" := FALSE;   // CH1.Alm.MinorFtcMouldOnLug.11 > CM1 outfeed buffer mould on lug sensor fault (1CM335BR9)
   Alm.MinorFtcMouldOnLug."12" := FALSE;   // CH1.Alm.MinorFtcMouldOnLug.12 > AC4 infeed mould on lug sensor fault (4AC330BR6)
   Alm.MinorFtcMouldOnLug."13" := FALSE;   // CH1.Alm.MinorFtcMouldOnLug.13 > AC4 outfeed mould on lug sensor fault (4AC430BR6)
   Alm.MinorFtcMouldOnLug."14" := FALSE;   // CH1.Alm.MinorFtcMouldOnLug.14 > OM1 outfeed mould on lug sensor fault (1OM333BR8)
   Alm.MinorFtcMouldOnLug."15" := FALSE;   // CH1.Alm.MinorFtcMouldOnLug.15 > RD1 infeed mould on lug sensor fault (1RD332BR3)
   Alm.MinorFtcMouldOnLug."16" := FALSE;   // CH1.Alm.MinorFtcMouldOnLug.16
   Alm.MinorFtcMouldOnLug."17" := FALSE;   // CH1.Alm.MinorFtcMouldOnLug.17
   Alm.MinorFtcMouldOnLug."18" := FALSE;   // CH1.Alm.MinorFtcMouldOnLug.18
   Alm.MinorFtcMouldOnLug."19" := FALSE;   // CH1.Alm.MinorFtcMouldOnLug.19
   Alm.MinorFtcMouldOnLug."20" := FALSE;   // CH1.Alm.MinorFtcMouldOnLug.20
   Alm.MinorFtcMouldOnLug."21" := FALSE;   // CH1.Alm.MinorFtcMouldOnLug.21
   Alm.MinorFtcMouldOnLug."22" := FALSE;   // CH1.Alm.MinorFtcMouldOnLug.22
   Alm.MinorFtcMouldOnLug."23" := FALSE;   // CH1.Alm.MinorFtcMouldOnLug.23
   Alm.MinorFtcMouldOnLug."24" := FALSE;   // CH1.Alm.MinorFtcMouldOnLug.24
   Alm.MinorFtcMouldOnLug."25" := FALSE;   // CH1.Alm.MinorFtcMouldOnLug.25
   Alm.MinorFtcMouldOnLug."26" := FALSE;   // CH1.Alm.MinorFtcMouldOnLug.26
   Alm.MinorFtcMouldOnLug."27" := FALSE;   // CH1.Alm.MinorFtcMouldOnLug.27
   Alm.MinorFtcMouldOnLug."28" := FALSE;   // CH1.Alm.MinorFtcMouldOnLug.28
   Alm.MinorFtcMouldOnLug."29" := FALSE;   // CH1.Alm.MinorFtcMouldOnLug.29
   Alm.MinorFtcMouldOnLug."30" := FALSE;   // CH1.Alm.MinorFtcMouldOnLug.30
   Alm.MinorFtcMouldOnLug."31" := FALSE;   // CH1.Alm.MinorFtcMouldOnLug.31
   Alm.MinorFtcMouldBtwAscDesc."0" := FALSE;   // CH1.Alm.MinorFtcMouldBtwAscDesc.0 > AC1 mould presence after battery 1 sensor fault (1AC330BR8)
   Alm.MinorFtcMouldBtwAscDesc."1" := FALSE;   // CH1.Alm.MinorFtcMouldBtwAscDesc.1 > AC2 mould presence after battery 1 sensor fault (2AC330BR8)
   Alm.MinorFtcMouldBtwAscDesc."2" := FALSE;   // CH1.Alm.MinorFtcMouldBtwAscDesc.2 > AC3 mould presence after battery 1 sensor fault (3AC330BR8)
   Alm.MinorFtcMouldBtwAscDesc."3" := FALSE;   // CH1.Alm.MinorFtcMouldBtwAscDesc.3 > AC4 mould presence after battery 1 sensor fault (4AC430BR8)
   Alm.MinorFtcMouldBtwAscDesc."4" := FALSE;   // CH1.Alm.MinorFtcMouldBtwAscDesc.4
   Alm.MinorFtcMouldBtwAscDesc."5" := FALSE;   // CH1.Alm.MinorFtcMouldBtwAscDesc.5
   Alm.MinorFtcMouldBtwAscDesc."6" := FALSE;   // CH1.Alm.MinorFtcMouldBtwAscDesc.6
   Alm.MinorFtcMouldBtwAscDesc."7" := FALSE;   // CH1.Alm.MinorFtcMouldBtwAscDesc.7
   Alm.MinorFtcMouldBtwAscDesc."8" := FALSE;   // CH1.Alm.MinorFtcMouldBtwAscDesc.8
   Alm.MinorFtcMouldBtwAscDesc."9" := FALSE;   // CH1.Alm.MinorFtcMouldBtwAscDesc.9
   Alm.MinorFtcMouldBtwAscDesc."10" := FALSE;   // CH1.Alm.MinorFtcMouldBtwAscDesc.10
   Alm.MinorFtcMouldBtwAscDesc."11" := FALSE;   // CH1.Alm.MinorFtcMouldBtwAscDesc.11
   Alm.MinorFtcMouldBtwAscDesc."12" := FALSE;   // CH1.Alm.MinorFtcMouldBtwAscDesc.12
   Alm.MinorFtcMouldBtwAscDesc."13" := FALSE;   // CH1.Alm.MinorFtcMouldBtwAscDesc.13
   Alm.MinorFtcMouldBtwAscDesc."14" := FALSE;   // CH1.Alm.MinorFtcMouldBtwAscDesc.14
   Alm.MinorFtcMouldBtwAscDesc."15" := FALSE;   // CH1.Alm.MinorFtcMouldBtwAscDesc.15
   Alm.MinorFtcMouldBtwAscDesc."16" := FALSE;   // CH1.Alm.MinorFtcMouldBtwAscDesc.16
   Alm.MinorFtcMouldBtwAscDesc."17" := FALSE;   // CH1.Alm.MinorFtcMouldBtwAscDesc.17
   Alm.MinorFtcMouldBtwAscDesc."18" := FALSE;   // CH1.Alm.MinorFtcMouldBtwAscDesc.18
   Alm.MinorFtcMouldBtwAscDesc."19" := FALSE;   // CH1.Alm.MinorFtcMouldBtwAscDesc.19
   Alm.MinorFtcMouldBtwAscDesc."20" := FALSE;   // CH1.Alm.MinorFtcMouldBtwAscDesc.20
   Alm.MinorFtcMouldBtwAscDesc."21" := FALSE;   // CH1.Alm.MinorFtcMouldBtwAscDesc.21
   Alm.MinorFtcMouldBtwAscDesc."22" := FALSE;   // CH1.Alm.MinorFtcMouldBtwAscDesc.22
   Alm.MinorFtcMouldBtwAscDesc."23" := FALSE;   // CH1.Alm.MinorFtcMouldBtwAscDesc.23
   Alm.MinorFtcMouldBtwAscDesc."24" := FALSE;   // CH1.Alm.MinorFtcMouldBtwAscDesc.24
   Alm.MinorFtcMouldBtwAscDesc."25" := FALSE;   // CH1.Alm.MinorFtcMouldBtwAscDesc.25
   Alm.MinorFtcMouldBtwAscDesc."26" := FALSE;   // CH1.Alm.MinorFtcMouldBtwAscDesc.26
   Alm.MinorFtcMouldBtwAscDesc."27" := FALSE;   // CH1.Alm.MinorFtcMouldBtwAscDesc.27
   Alm.MinorFtcMouldBtwAscDesc."28" := FALSE;   // CH1.Alm.MinorFtcMouldBtwAscDesc.28
   Alm.MinorFtcMouldBtwAscDesc."29" := FALSE;   // CH1.Alm.MinorFtcMouldBtwAscDesc.29
   Alm.MinorFtcMouldBtwAscDesc."30" := FALSE;   // CH1.Alm.MinorFtcMouldBtwAscDesc.30
   Alm.MinorFtcMouldBtwAscDesc."31" := FALSE;   // CH1.Alm.MinorFtcMouldBtwAscDesc.31
   Alm.MinorChain1."0" := FALSE;   // CH1.Alm.MinorChain1.0
   Alm.MinorChain1."1" := FALSE;   // CH1.Alm.MinorChain1.1
   Alm.MinorChain1."2" := FALSE;   // CH1.Alm.MinorChain1.2
   Alm.MinorChain1."3" := FALSE;   // CH1.Alm.MinorChain1.3 > Chain 1 torque limit (1CH40MA8)
   Alm.MinorChain1."4" := FALSE;   // CH1.Alm.MinorChain1.4 > Chain 1 drive fault (1CH40MA8)
   Alm.MinorChain1."5" := FALSE;   // CH1.Alm.MinorChain1.5 > Chain 1 loss of zero position (1CH40MA8)
   Alm.MinorChain1."6" := FALSE;   // CH1.Alm.MinorChain1.6
   Alm.MinorChain1."7" := FALSE;   // CH1.Alm.MinorChain1.7 > Chain 1 safety not ok sinamics (1CH40MA8)
   Alm.MinorChain1."8" := FALSE;   // CH1.Alm.MinorChain1.8 > Chain 1 not in phase (1CH40MA8)
   Alm.MinorChain1."9" := FALSE;   // CH1.Alm.MinorChain1.9 > Chain 1 obstruction - mould presence end chain (1CH40MA8)
   Alm.MinorChain1."10" := FALSE;   // CH1.Alm.MinorChain1.10 > Chain 1 waiting for operator validation
   Alm.MinorChain1."11" := FALSE;   // CH1.Alm.MinorChain1.11 > Chain 1 slave forward refer to master
   Alm.MinorChain1."12" := FALSE;   // CH1.Alm.MinorChain1.12 > Chain 1 slave backward refer to master
   Alm.MinorChain1."13" := FALSE;   // CH1.Alm.MinorChain1.13 > Chain 1 slave unwind refer to master
   Alm.MinorChain1."14" := FALSE;   // CH1.Alm.MinorChain1.14 > Chain 1 error cam hooking
   Alm.MinorChain1."15" := FALSE;   // CH1.Alm.MinorChain1.15
   Alm.MinorChain1."16" := FALSE;   // CH1.Alm.MinorChain1.16
   Alm.MinorChain1."17" := FALSE;   // CH1.Alm.MinorChain1.17
   Alm.MinorChain1."18" := FALSE;   // CH1.Alm.MinorChain1.18
   Alm.MinorChain1."19" := FALSE;   // CH1.Alm.MinorChain1.19
   Alm.MinorChain1."20" := FALSE;   // CH1.Alm.MinorChain1.20
   Alm.MinorChain1."21" := FALSE;   // CH1.Alm.MinorChain1.21
   Alm.MinorChain1."22" := FALSE;   // CH1.Alm.MinorChain1.22
   Alm.MinorChain1."23" := FALSE;   // CH1.Alm.MinorChain1.23
   Alm.MinorChain1."24" := FALSE;   // CH1.Alm.MinorChain1.24
   Alm.MinorChain1."25" := FALSE;   // CH1.Alm.MinorChain1.25
   Alm.MinorChain1."26" := FALSE;   // CH1.Alm.MinorChain1.26
   Alm.MinorChain1."27" := FALSE;   // CH1.Alm.MinorChain1.27
   Alm.MinorChain1."28" := FALSE;   // CH1.Alm.MinorChain1.28
   Alm.MinorChain1."29" := FALSE;   // CH1.Alm.MinorChain1.29
   Alm.MinorChain1."30" := FALSE;   // CH1.Alm.MinorChain1.30
   Alm.MinorChain1."31" := FALSE;   // CH1.Alm.MinorChain1.31
   Alm.MinorChain2."0" := FALSE;   // CH1.Alm.MinorChain2.0
   Alm.MinorChain2."1" := FALSE;   // CH1.Alm.MinorChain2.1
   Alm.MinorChain2."2" := FALSE;   // CH1.Alm.MinorChain2.2
   Alm.MinorChain2."3" := FALSE;   // CH1.Alm.MinorChain2.3 > Chain 2 torque limit (1CH41MA8)
   Alm.MinorChain2."4" := FALSE;   // CH1.Alm.MinorChain2.4 > Chain 2 drive fault (1CH41MA8)
   Alm.MinorChain2."5" := FALSE;   // CH1.Alm.MinorChain2.5 > Chain 2 loss of zero position (1CH41MA8)
   Alm.MinorChain2."6" := FALSE;   // CH1.Alm.MinorChain2.6
   Alm.MinorChain2."7" := FALSE;   // CH1.Alm.MinorChain2.7 > Chain 2 safety not ok sinamics (1CH41MA8)
   Alm.MinorChain2."8" := FALSE;   // CH1.Alm.MinorChain2.8 > Chain 2 not in phase (1CH41MA8)
   Alm.MinorChain2."9" := FALSE;   // CH1.Alm.MinorChain2.9 > Chain 2 obstruction - mould presence end chain (1CH41MA8)
   Alm.MinorChain2."10" := FALSE;   // CH1.Alm.MinorChain2.10 > Chain 2 waiting for operator validation
   Alm.MinorChain2."11" := FALSE;   // CH1.Alm.MinorChain2.11 > Chain 2 slave forward refer to master
   Alm.MinorChain2."12" := FALSE;   // CH1.Alm.MinorChain2.12 > Chain 2 slave backward refer to master
   Alm.MinorChain2."13" := FALSE;   // CH1.Alm.MinorChain2.13 > Chain 2 slave unwind refer to master
   Alm.MinorChain2."14" := FALSE;   // CH1.Alm.MinorChain2.14 > Chain 2 error cam hooking
   Alm.MinorChain2."15" := FALSE;   // CH1.Alm.MinorChain2.15
   Alm.MinorChain2."16" := FALSE;   // CH1.Alm.MinorChain2.16
   Alm.MinorChain2."17" := FALSE;   // CH1.Alm.MinorChain2.17
   Alm.MinorChain2."18" := FALSE;   // CH1.Alm.MinorChain2.18
   Alm.MinorChain2."19" := FALSE;   // CH1.Alm.MinorChain2.19
   Alm.MinorChain2."20" := FALSE;   // CH1.Alm.MinorChain2.20
   Alm.MinorChain2."21" := FALSE;   // CH1.Alm.MinorChain2.21
   Alm.MinorChain2."22" := FALSE;   // CH1.Alm.MinorChain2.22
   Alm.MinorChain2."23" := FALSE;   // CH1.Alm.MinorChain2.23
   Alm.MinorChain2."24" := FALSE;   // CH1.Alm.MinorChain2.24
   Alm.MinorChain2."25" := FALSE;   // CH1.Alm.MinorChain2.25
   Alm.MinorChain2."26" := FALSE;   // CH1.Alm.MinorChain2.26
   Alm.MinorChain2."27" := FALSE;   // CH1.Alm.MinorChain2.27
   Alm.MinorChain2."28" := FALSE;   // CH1.Alm.MinorChain2.28
   Alm.MinorChain2."29" := FALSE;   // CH1.Alm.MinorChain2.29
   Alm.MinorChain2."30" := FALSE;   // CH1.Alm.MinorChain2.30
   Alm.MinorChain2."31" := FALSE;   // CH1.Alm.MinorChain2.31
   Alm.MinorChain3."0" := FALSE;   // CH1.Alm.MinorChain3.0
   Alm.MinorChain3."1" := FALSE;   // CH1.Alm.MinorChain3.1
   Alm.MinorChain3."2" := FALSE;   // CH1.Alm.MinorChain3.2
   Alm.MinorChain3."3" := FALSE;   // CH1.Alm.MinorChain3.3 > Chain 3 torque limit (1CH42MA8)
   Alm.MinorChain3."4" := FALSE;   // CH1.Alm.MinorChain3.4 > Chain 3 drive fault (1CH42MA8)
   Alm.MinorChain3."5" := FALSE;   // CH1.Alm.MinorChain3.5 > Chain 3 loss of zero position (1CH42MA8)
   Alm.MinorChain3."6" := FALSE;   // CH1.Alm.MinorChain3.6
   Alm.MinorChain3."7" := FALSE;   // CH1.Alm.MinorChain3.7 > Chain 3 safety not ok sinamics (1CH42MA8)
   Alm.MinorChain3."8" := FALSE;   // CH1.Alm.MinorChain3.8 > Chain 3 not in phase (1CH42MA8)
   Alm.MinorChain3."9" := FALSE;   // CH1.Alm.MinorChain3.9 > Chain 3 obstruction - mould presence end chain (1CH42MA8)
   Alm.MinorChain3."10" := FALSE;   // CH1.Alm.MinorChain3.10 > Chain 3 waiting for operator validation
   Alm.MinorChain3."11" := FALSE;   // CH1.Alm.MinorChain3.11 > Chain 3 slave forward refer to master
   Alm.MinorChain3."12" := FALSE;   // CH1.Alm.MinorChain3.12 > Chain 3 slave backward refer to master
   Alm.MinorChain3."13" := FALSE;   // CH1.Alm.MinorChain3.13 > Chain 3 slave unwind refer to master
   Alm.MinorChain3."14" := FALSE;   // CH1.Alm.MinorChain3.14 > Chain 3 error cam hooking
   Alm.MinorChain3."15" := FALSE;   // CH1.Alm.MinorChain3.15
   Alm.MinorChain3."16" := FALSE;   // CH1.Alm.MinorChain3.16
   Alm.MinorChain3."17" := FALSE;   // CH1.Alm.MinorChain3.17
   Alm.MinorChain3."18" := FALSE;   // CH1.Alm.MinorChain3.18
   Alm.MinorChain3."19" := FALSE;   // CH1.Alm.MinorChain3.19
   Alm.MinorChain3."20" := FALSE;   // CH1.Alm.MinorChain3.20
   Alm.MinorChain3."21" := FALSE;   // CH1.Alm.MinorChain3.21
   Alm.MinorChain3."22" := FALSE;   // CH1.Alm.MinorChain3.22
   Alm.MinorChain3."23" := FALSE;   // CH1.Alm.MinorChain3.23
   Alm.MinorChain3."24" := FALSE;   // CH1.Alm.MinorChain3.24
   Alm.MinorChain3."25" := FALSE;   // CH1.Alm.MinorChain3.25
   Alm.MinorChain3."26" := FALSE;   // CH1.Alm.MinorChain3.26
   Alm.MinorChain3."27" := FALSE;   // CH1.Alm.MinorChain3.27
   Alm.MinorChain3."28" := FALSE;   // CH1.Alm.MinorChain3.28
   Alm.MinorChain3."29" := FALSE;   // CH1.Alm.MinorChain3.29
   Alm.MinorChain3."30" := FALSE;   // CH1.Alm.MinorChain3.30
   Alm.MinorChain3."31" := FALSE;   // CH1.Alm.MinorChain3.31
   Alm.MinorChain4."0" := FALSE;   // CH1.Alm.MinorChain4.0
   Alm.MinorChain4."1" := FALSE;   // CH1.Alm.MinorChain4.1
   Alm.MinorChain4."2" := FALSE;   // CH1.Alm.MinorChain4.2
   Alm.MinorChain4."3" := FALSE;   // CH1.Alm.MinorChain4.3 > Chain 4 torque limit (1CH44MA8)
   Alm.MinorChain4."4" := FALSE;   // CH1.Alm.MinorChain4.4 > Chain 4 drive fault (1CH44MA8)
   Alm.MinorChain4."5" := FALSE;   // CH1.Alm.MinorChain4.5 > Chain 4 loss of zero position (1CH44MA8)
   Alm.MinorChain4."6" := FALSE;   // CH1.Alm.MinorChain4.6
   Alm.MinorChain4."7" := FALSE;   // CH1.Alm.MinorChain4.7 > Chain 4 safety not ok sinamics (1CH44MA8)
   Alm.MinorChain4."8" := FALSE;   // CH1.Alm.MinorChain4.8 > Chain 4 not in phase (1CH44MA8)
   Alm.MinorChain4."9" := FALSE;   // CH1.Alm.MinorChain4.9 > Chain 4 obstruction - mould presence end chain (1CH44MA8)
   Alm.MinorChain4."10" := FALSE;   // CH1.Alm.MinorChain4.10 > Chain 4 waiting for operator validation
   Alm.MinorChain4."11" := FALSE;   // CH1.Alm.MinorChain4.11 > Chain 4 slave forward refer to master
   Alm.MinorChain4."12" := FALSE;   // CH1.Alm.MinorChain4.12 > Chain 4 slave backward refer to master
   Alm.MinorChain4."13" := FALSE;   // CH1.Alm.MinorChain4.13 > Chain 4 slave unwind refer to master
   Alm.MinorChain4."14" := FALSE;   // CH1.Alm.MinorChain4.14 > Chain 4 error cam hooking
   Alm.MinorChain4."15" := FALSE;   // CH1.Alm.MinorChain4.15
   Alm.MinorChain4."16" := FALSE;   // CH1.Alm.MinorChain4.16
   Alm.MinorChain4."17" := FALSE;   // CH1.Alm.MinorChain4.17
   Alm.MinorChain4."18" := FALSE;   // CH1.Alm.MinorChain4.18
   Alm.MinorChain4."19" := FALSE;   // CH1.Alm.MinorChain4.19
   Alm.MinorChain4."20" := FALSE;   // CH1.Alm.MinorChain4.20
   Alm.MinorChain4."21" := FALSE;   // CH1.Alm.MinorChain4.21
   Alm.MinorChain4."22" := FALSE;   // CH1.Alm.MinorChain4.22
   Alm.MinorChain4."23" := FALSE;   // CH1.Alm.MinorChain4.23
   Alm.MinorChain4."24" := FALSE;   // CH1.Alm.MinorChain4.24
   Alm.MinorChain4."25" := FALSE;   // CH1.Alm.MinorChain4.25
   Alm.MinorChain4."26" := FALSE;   // CH1.Alm.MinorChain4.26
   Alm.MinorChain4."27" := FALSE;   // CH1.Alm.MinorChain4.27
   Alm.MinorChain4."28" := FALSE;   // CH1.Alm.MinorChain4.28
   Alm.MinorChain4."29" := FALSE;   // CH1.Alm.MinorChain4.29
   Alm.MinorChain4."30" := FALSE;   // CH1.Alm.MinorChain4.30
   Alm.MinorChain4."31" := FALSE;   // CH1.Alm.MinorChain4.31
   Alm.MinorChain5."0" := FALSE;   // CH1.Alm.MinorChain5.0
   Alm.MinorChain5."1" := FALSE;   // CH1.Alm.MinorChain5.1
   Alm.MinorChain5."2" := FALSE;   // CH1.Alm.MinorChain5.2
   Alm.MinorChain5."3" := FALSE;   // CH1.Alm.MinorChain5.3 > Chain 5 torque limit (1CH48MA8)
   Alm.MinorChain5."4" := FALSE;   // CH1.Alm.MinorChain5.4 > Chain 5 drive fault (1CH48MA8)
   Alm.MinorChain5."5" := FALSE;   // CH1.Alm.MinorChain5.5 > Chain 5 loss of zero position (1CH48MA8)
   Alm.MinorChain5."6" := FALSE;   // CH1.Alm.MinorChain5.6
   Alm.MinorChain5."7" := FALSE;   // CH1.Alm.MinorChain5.7 > Chain 5 safety not ok sinamics (1CH48MA8)
   Alm.MinorChain5."8" := FALSE;   // CH1.Alm.MinorChain5.8 > Chain 5 not in phase (1CH48MA8)
   Alm.MinorChain5."9" := FALSE;   // CH1.Alm.MinorChain5.9 > Chain 5 obstruction - mould presence end chain (1CH48MA8)
   Alm.MinorChain5."10" := FALSE;   // CH1.Alm.MinorChain5.10 > Chain 5 waiting for operator validation
   Alm.MinorChain5."11" := FALSE;   // CH1.Alm.MinorChain5.11 > Chain 5 slave forward refer to master
   Alm.MinorChain5."12" := FALSE;   // CH1.Alm.MinorChain5.12 > Chain 5 slave backward refer to master
   Alm.MinorChain5."13" := FALSE;   // CH1.Alm.MinorChain5.13 > Chain 5 slave unwind refer to master
   Alm.MinorChain5."14" := FALSE;   // CH1.Alm.MinorChain5.14 > Chain 5 error cam hooking
   Alm.MinorChain5."15" := FALSE;   // CH1.Alm.MinorChain5.15
   Alm.MinorChain5."16" := FALSE;   // CH1.Alm.MinorChain5.16
   Alm.MinorChain5."17" := FALSE;   // CH1.Alm.MinorChain5.17
   Alm.MinorChain5."18" := FALSE;   // CH1.Alm.MinorChain5.18
   Alm.MinorChain5."19" := FALSE;   // CH1.Alm.MinorChain5.19
   Alm.MinorChain5."20" := FALSE;   // CH1.Alm.MinorChain5.20
   Alm.MinorChain5."21" := FALSE;   // CH1.Alm.MinorChain5.21
   Alm.MinorChain5."22" := FALSE;   // CH1.Alm.MinorChain5.22
   Alm.MinorChain5."23" := FALSE;   // CH1.Alm.MinorChain5.23
   Alm.MinorChain5."24" := FALSE;   // CH1.Alm.MinorChain5.24
   Alm.MinorChain5."25" := FALSE;   // CH1.Alm.MinorChain5.25
   Alm.MinorChain5."26" := FALSE;   // CH1.Alm.MinorChain5.26
   Alm.MinorChain5."27" := FALSE;   // CH1.Alm.MinorChain5.27
   Alm.MinorChain5."28" := FALSE;   // CH1.Alm.MinorChain5.28
   Alm.MinorChain5."29" := FALSE;   // CH1.Alm.MinorChain5.29
   Alm.MinorChain5."30" := FALSE;   // CH1.Alm.MinorChain5.30
   Alm.MinorChain5."31" := FALSE;   // CH1.Alm.MinorChain5.31
   Alm.MinorChain6."0" := FALSE;   // CH1.Alm.MinorChain6.0
   Alm.MinorChain6."1" := FALSE;   // CH1.Alm.MinorChain6.1
   Alm.MinorChain6."2" := FALSE;   // CH1.Alm.MinorChain6.2
   Alm.MinorChain6."3" := FALSE;   // CH1.Alm.MinorChain6.3 > Chain 6 torque limit (1CH46MA8)
   Alm.MinorChain6."4" := FALSE;   // CH1.Alm.MinorChain6.4 > Chain 6 drive fault (1CH46MA8)
   Alm.MinorChain6."5" := FALSE;   // CH1.Alm.MinorChain6.5 > Chain 6 loss of zero position (1CH46MA8)
   Alm.MinorChain6."6" := FALSE;   // CH1.Alm.MinorChain6.6
   Alm.MinorChain6."7" := FALSE;   // CH1.Alm.MinorChain6.7 > Chain 6 safety not ok sinamics (1CH46MA8)
   Alm.MinorChain6."8" := FALSE;   // CH1.Alm.MinorChain6.8 > Chain 6 not in phase (1CH46MA8)
   Alm.MinorChain6."9" := FALSE;   // CH1.Alm.MinorChain6.9 > Chain 6 obstruction - mould presence end chain (1CH46MA8)
   Alm.MinorChain6."10" := FALSE;   // CH1.Alm.MinorChain6.10 > Chain 6 waiting for operator validation
   Alm.MinorChain6."11" := FALSE;   // CH1.Alm.MinorChain6.11 > Chain 6 slave forward refer to master
   Alm.MinorChain6."12" := FALSE;   // CH1.Alm.MinorChain6.12 > Chain 6 slave backward refer to master
   Alm.MinorChain6."13" := FALSE;   // CH1.Alm.MinorChain6.13 > Chain 6 slave unwind refer to master
   Alm.MinorChain6."14" := FALSE;   // CH1.Alm.MinorChain6.14 > Chain 6 error cam hooking
   Alm.MinorChain6."15" := FALSE;   // CH1.Alm.MinorChain6.15
   Alm.MinorChain6."16" := FALSE;   // CH1.Alm.MinorChain6.16
   Alm.MinorChain6."17" := FALSE;   // CH1.Alm.MinorChain6.17
   Alm.MinorChain6."18" := FALSE;   // CH1.Alm.MinorChain6.18
   Alm.MinorChain6."19" := FALSE;   // CH1.Alm.MinorChain6.19
   Alm.MinorChain6."20" := FALSE;   // CH1.Alm.MinorChain6.20
   Alm.MinorChain6."21" := FALSE;   // CH1.Alm.MinorChain6.21
   Alm.MinorChain6."22" := FALSE;   // CH1.Alm.MinorChain6.22
   Alm.MinorChain6."23" := FALSE;   // CH1.Alm.MinorChain6.23
   Alm.MinorChain6."24" := FALSE;   // CH1.Alm.MinorChain6.24
   Alm.MinorChain6."25" := FALSE;   // CH1.Alm.MinorChain6.25
   Alm.MinorChain6."26" := FALSE;   // CH1.Alm.MinorChain6.26
   Alm.MinorChain6."27" := FALSE;   // CH1.Alm.MinorChain6.27
   Alm.MinorChain6."28" := FALSE;   // CH1.Alm.MinorChain6.28
   Alm.MinorChain6."29" := FALSE;   // CH1.Alm.MinorChain6.29
   Alm.MinorChain6."30" := FALSE;   // CH1.Alm.MinorChain6.30
   Alm.MinorChain6."31" := FALSE;   // CH1.Alm.MinorChain6.31
   Alm.MinorChain7."0" := FALSE;   // CH1.Alm.MinorChain7.0
   Alm.MinorChain7."1" := FALSE;   // CH1.Alm.MinorChain7.1
   Alm.MinorChain7."2" := FALSE;   // CH1.Alm.MinorChain7.2
   Alm.MinorChain7."3" := FALSE;   // CH1.Alm.MinorChain7.3 > Chain 7 torque limit (1CH49MA8)
   Alm.MinorChain7."4" := FALSE;   // CH1.Alm.MinorChain7.4 > Chain 7 drive fault (1CH49MA8)
   Alm.MinorChain7."5" := FALSE;   // CH1.Alm.MinorChain7.5 > Chain 7 loss of zero position (1CH49MA8)
   Alm.MinorChain7."6" := FALSE;   // CH1.Alm.MinorChain7.6
   Alm.MinorChain7."7" := FALSE;   // CH1.Alm.MinorChain7.7 > Chain 7 safety not ok sinamics (1CH49MA8)
   Alm.MinorChain7."8" := FALSE;   // CH1.Alm.MinorChain7.8 > Chain 7 not in phase (1CH49MA8)
   Alm.MinorChain7."9" := FALSE;   // CH1.Alm.MinorChain7.9 > Chain 7 obstruction - mould presence end chain (1CH49MA8)
   Alm.MinorChain7."10" := FALSE;   // CH1.Alm.MinorChain7.10 > Chain 7 waiting for operator validation
   Alm.MinorChain7."11" := FALSE;   // CH1.Alm.MinorChain7.11 > Chain 7 slave forward refer to master
   Alm.MinorChain7."12" := FALSE;   // CH1.Alm.MinorChain7.12 > Chain 7 slave backward refer to master
   Alm.MinorChain7."13" := FALSE;   // CH1.Alm.MinorChain7.13 > Chain 7 slave unwind refer to master
   Alm.MinorChain7."14" := FALSE;   // CH1.Alm.MinorChain7.14 > Chain 7 error cam hooking
   Alm.MinorChain7."15" := FALSE;   // CH1.Alm.MinorChain7.15
   Alm.MinorChain7."16" := FALSE;   // CH1.Alm.MinorChain7.16
   Alm.MinorChain7."17" := FALSE;   // CH1.Alm.MinorChain7.17
   Alm.MinorChain7."18" := FALSE;   // CH1.Alm.MinorChain7.18
   Alm.MinorChain7."19" := FALSE;   // CH1.Alm.MinorChain7.19
   Alm.MinorChain7."20" := FALSE;   // CH1.Alm.MinorChain7.20
   Alm.MinorChain7."21" := FALSE;   // CH1.Alm.MinorChain7.21
   Alm.MinorChain7."22" := FALSE;   // CH1.Alm.MinorChain7.22
   Alm.MinorChain7."23" := FALSE;   // CH1.Alm.MinorChain7.23
   Alm.MinorChain7."24" := FALSE;   // CH1.Alm.MinorChain7.24
   Alm.MinorChain7."25" := FALSE;   // CH1.Alm.MinorChain7.25
   Alm.MinorChain7."26" := FALSE;   // CH1.Alm.MinorChain7.26
   Alm.MinorChain7."27" := FALSE;   // CH1.Alm.MinorChain7.27
   Alm.MinorChain7."28" := FALSE;   // CH1.Alm.MinorChain7.28
   Alm.MinorChain7."29" := FALSE;   // CH1.Alm.MinorChain7.29
   Alm.MinorChain7."30" := FALSE;   // CH1.Alm.MinorChain7.30
   Alm.MinorChain7."31" := FALSE;   // CH1.Alm.MinorChain7.31
   Alm.MinorChain8."0" := FALSE;   // CH1.Alm.MinorChain8.0
   Alm.MinorChain8."1" := FALSE;   // CH1.Alm.MinorChain8.1
   Alm.MinorChain8."2" := FALSE;   // CH1.Alm.MinorChain8.2
   Alm.MinorChain8."3" := FALSE;   // CH1.Alm.MinorChain8.3 > Chain 8 torque limit (1CH45MA8)
   Alm.MinorChain8."4" := FALSE;   // CH1.Alm.MinorChain8.4 > Chain 8 drive fault (1CH45MA8)
   Alm.MinorChain8."5" := FALSE;   // CH1.Alm.MinorChain8.5 > Chain 8 loss of zero position (1CH45MA8)
   Alm.MinorChain8."6" := FALSE;   // CH1.Alm.MinorChain8.6
   Alm.MinorChain8."7" := FALSE;   // CH1.Alm.MinorChain8.7 > Chain 8 safety not ok sinamics (1CH45MA8)
   Alm.MinorChain8."8" := FALSE;   // CH1.Alm.MinorChain8.8 > Chain 8 not in phase (1CH45MA8)
   Alm.MinorChain8."9" := FALSE;   // CH1.Alm.MinorChain8.9 > Chain 8 obstruction - mould presence end chain (1CH45MA8)
   Alm.MinorChain8."10" := FALSE;   // CH1.Alm.MinorChain8.10 > Chain 8 waiting for operator validation
   Alm.MinorChain8."11" := FALSE;   // CH1.Alm.MinorChain8.11 > Chain 8 slave forward refer to master
   Alm.MinorChain8."12" := FALSE;   // CH1.Alm.MinorChain8.12 > Chain 8 slave backward refer to master
   Alm.MinorChain8."13" := FALSE;   // CH1.Alm.MinorChain8.13 > Chain 8 slave unwind refer to master
   Alm.MinorChain8."14" := FALSE;   // CH1.Alm.MinorChain8.14 > Chain 8 error cam hooking
   Alm.MinorChain8."15" := FALSE;   // CH1.Alm.MinorChain8.15
   Alm.MinorChain8."16" := FALSE;   // CH1.Alm.MinorChain8.16
   Alm.MinorChain8."17" := FALSE;   // CH1.Alm.MinorChain8.17
   Alm.MinorChain8."18" := FALSE;   // CH1.Alm.MinorChain8.18
   Alm.MinorChain8."19" := FALSE;   // CH1.Alm.MinorChain8.19
   Alm.MinorChain8."20" := FALSE;   // CH1.Alm.MinorChain8.20
   Alm.MinorChain8."21" := FALSE;   // CH1.Alm.MinorChain8.21
   Alm.MinorChain8."22" := FALSE;   // CH1.Alm.MinorChain8.22
   Alm.MinorChain8."23" := FALSE;   // CH1.Alm.MinorChain8.23
   Alm.MinorChain8."24" := FALSE;   // CH1.Alm.MinorChain8.24
   Alm.MinorChain8."25" := FALSE;   // CH1.Alm.MinorChain8.25
   Alm.MinorChain8."26" := FALSE;   // CH1.Alm.MinorChain8.26
   Alm.MinorChain8."27" := FALSE;   // CH1.Alm.MinorChain8.27
   Alm.MinorChain8."28" := FALSE;   // CH1.Alm.MinorChain8.28
   Alm.MinorChain8."29" := FALSE;   // CH1.Alm.MinorChain8.29
   Alm.MinorChain8."30" := FALSE;   // CH1.Alm.MinorChain8.30
   Alm.MinorChain8."31" := FALSE;   // CH1.Alm.MinorChain8.31
   Sign.General."0" := FALSE;   // CH1.Sign.General.0
   Sign.General."1" := FALSE;   // CH1.Sign.General.1
   Sign.General."2" := FALSE;   // CH1.Sign.General.2
   Sign.General."3" := FALSE;   // CH1.Sign.General.3
   Sign.General."4" := FALSE;   // CH1.Sign.General.4
   Sign.General."5" := FALSE;   // CH1.Sign.General.5
   Sign.General."6" := FALSE;   // CH1.Sign.General.6
   Sign.General."7" := FALSE;   // CH1.Sign.General.7
   Sign.General."8" := FALSE;   // CH1.Sign.General.8
   Sign.General."9" := FALSE;   // CH1.Sign.General.9
   Sign.General."10" := FALSE;   // CH1.Sign.General.10
   Sign.General."11" := FALSE;   // CH1.Sign.General.11
   Sign.General."12" := FALSE;   // CH1.Sign.General.12
   Sign.General."13" := FALSE;   // CH1.Sign.General.13
   Sign.General."14" := FALSE;   // CH1.Sign.General.14
   Sign.General."15" := FALSE;   // CH1.Sign.General.15
   Sign.General."16" := FALSE;   // CH1.Sign.General.16
   Sign.General."17" := FALSE;   // CH1.Sign.General.17
   Sign.General."18" := FALSE;   // CH1.Sign.General.18
   Sign.General."19" := FALSE;   // CH1.Sign.General.19
   Sign.General."20" := FALSE;   // CH1.Sign.General.20
   Sign.General."21" := FALSE;   // CH1.Sign.General.21
   Sign.General."22" := FALSE;   // CH1.Sign.General.22
   Sign.General."23" := FALSE;   // CH1.Sign.General.23
   Sign.General."24" := FALSE;   // CH1.Sign.General.24
   Sign.General."25" := FALSE;   // CH1.Sign.General.25
   Sign.General."26" := FALSE;   // CH1.Sign.General.26
   Sign.General."27" := FALSE;   // CH1.Sign.General.27
   Sign.General."28" := FALSE;   // CH1.Sign.General.28
   Sign.General."29" := FALSE;   // CH1.Sign.General.29
   Sign.General."30" := FALSE;   // CH1.Sign.General.30
   Sign.General."31" := FALSE;   // CH1.Sign.General.31
   Sign.Maintenance_Req."0" := FALSE;   // CH1.Sign.Maintenance_Req.0 > Maintenance 0 request
   Sign.Maintenance_Req."1" := FALSE;   // CH1.Sign.Maintenance_Req.1 > Maintenance 1 request
   Sign.Maintenance_Req."2" := FALSE;   // CH1.Sign.Maintenance_Req.2 > Maintenance 2 request
   Sign.Maintenance_Req."3" := FALSE;   // CH1.Sign.Maintenance_Req.3 > Maintenance 3 request
   Sign.Maintenance_Req."4" := FALSE;   // CH1.Sign.Maintenance_Req.4 > Maintenance 4 request
   Sign.Maintenance_Req."5" := FALSE;   // CH1.Sign.Maintenance_Req.5 > Maintenance 5 request
   Sign.Maintenance_Req."6" := FALSE;   // CH1.Sign.Maintenance_Req.6 > Maintenance 6 request
   Sign.Maintenance_Req."7" := FALSE;   // CH1.Sign.Maintenance_Req.7 > Maintenance 7 request
   Sign.Maintenance_Req."8" := FALSE;   // CH1.Sign.Maintenance_Req.8 > Maintenance 8 request
   Sign.Maintenance_Req."9" := FALSE;   // CH1.Sign.Maintenance_Req.9 > Maintenance 9 request
   Sign.Maintenance_Req."10" := FALSE;   // CH1.Sign.Maintenance_Req.10
   Sign.Maintenance_Req."11" := FALSE;   // CH1.Sign.Maintenance_Req.11
   Sign.Maintenance_Req."12" := FALSE;   // CH1.Sign.Maintenance_Req.12
   Sign.Maintenance_Req."13" := FALSE;   // CH1.Sign.Maintenance_Req.13
   Sign.Maintenance_Req."14" := FALSE;   // CH1.Sign.Maintenance_Req.14
   Sign.Maintenance_Req."15" := FALSE;   // CH1.Sign.Maintenance_Req.15
   Sign.Maintenance_Req."16" := FALSE;   // CH1.Sign.Maintenance_Req.16
   Sign.Maintenance_Req."17" := FALSE;   // CH1.Sign.Maintenance_Req.17
   Sign.Maintenance_Req."18" := FALSE;   // CH1.Sign.Maintenance_Req.18
   Sign.Maintenance_Req."19" := FALSE;   // CH1.Sign.Maintenance_Req.19
   Sign.Maintenance_Req."20" := FALSE;   // CH1.Sign.Maintenance_Req.20
   Sign.Maintenance_Req."21" := FALSE;   // CH1.Sign.Maintenance_Req.21
   Sign.Maintenance_Req."22" := FALSE;   // CH1.Sign.Maintenance_Req.22
   Sign.Maintenance_Req."23" := FALSE;   // CH1.Sign.Maintenance_Req.23
   Sign.Maintenance_Req."24" := FALSE;   // CH1.Sign.Maintenance_Req.24
   Sign.Maintenance_Req."25" := FALSE;   // CH1.Sign.Maintenance_Req.25
   Sign.Maintenance_Req."26" := FALSE;   // CH1.Sign.Maintenance_Req.26
   Sign.Maintenance_Req."27" := FALSE;   // CH1.Sign.Maintenance_Req.27
   Sign.Maintenance_Req."28" := FALSE;   // CH1.Sign.Maintenance_Req.28
   Sign.Maintenance_Req."29" := FALSE;   // CH1.Sign.Maintenance_Req.29
   Sign.Maintenance_Req."30" := FALSE;   // CH1.Sign.Maintenance_Req.30
   Sign.Maintenance_Req."31" := FALSE;   // CH1.Sign.Maintenance_Req.31
   Sign.Maintenance_Activated."0" := FALSE;   // CH1.Sign.Maintenance_Activated.0 > Maintenance 0 activated
   Sign.Maintenance_Activated."1" := FALSE;   // CH1.Sign.Maintenance_Activated.1 > Maintenance 1 activated
   Sign.Maintenance_Activated."2" := FALSE;   // CH1.Sign.Maintenance_Activated.2 > Maintenance 2 activated
   Sign.Maintenance_Activated."3" := FALSE;   // CH1.Sign.Maintenance_Activated.3 > Maintenance 3 activated
   Sign.Maintenance_Activated."4" := FALSE;   // CH1.Sign.Maintenance_Activated.4 > Maintenance 4 activated
   Sign.Maintenance_Activated."5" := FALSE;   // CH1.Sign.Maintenance_Activated.5 > Maintenance 5 activated
   Sign.Maintenance_Activated."6" := FALSE;   // CH1.Sign.Maintenance_Activated.6 > Maintenance 6 activated
   Sign.Maintenance_Activated."7" := FALSE;   // CH1.Sign.Maintenance_Activated.7 > Maintenance 7 activated
   Sign.Maintenance_Activated."8" := FALSE;   // CH1.Sign.Maintenance_Activated.8 > Maintenance 8 activated
   Sign.Maintenance_Activated."9" := FALSE;   // CH1.Sign.Maintenance_Activated.9 > Maintenance 9 activated
   Sign.Maintenance_Activated."10" := FALSE;   // CH1.Sign.Maintenance_Activated.10
   Sign.Maintenance_Activated."11" := FALSE;   // CH1.Sign.Maintenance_Activated.11
   Sign.Maintenance_Activated."12" := FALSE;   // CH1.Sign.Maintenance_Activated.12
   Sign.Maintenance_Activated."13" := FALSE;   // CH1.Sign.Maintenance_Activated.13
   Sign.Maintenance_Activated."14" := FALSE;   // CH1.Sign.Maintenance_Activated.14
   Sign.Maintenance_Activated."15" := FALSE;   // CH1.Sign.Maintenance_Activated.15
   Sign.Maintenance_Activated."16" := FALSE;   // CH1.Sign.Maintenance_Activated.16
   Sign.Maintenance_Activated."17" := FALSE;   // CH1.Sign.Maintenance_Activated.17
   Sign.Maintenance_Activated."18" := FALSE;   // CH1.Sign.Maintenance_Activated.18
   Sign.Maintenance_Activated."19" := FALSE;   // CH1.Sign.Maintenance_Activated.19
   Sign.Maintenance_Activated."20" := FALSE;   // CH1.Sign.Maintenance_Activated.20
   Sign.Maintenance_Activated."21" := FALSE;   // CH1.Sign.Maintenance_Activated.21
   Sign.Maintenance_Activated."22" := FALSE;   // CH1.Sign.Maintenance_Activated.22
   Sign.Maintenance_Activated."23" := FALSE;   // CH1.Sign.Maintenance_Activated.23
   Sign.Maintenance_Activated."24" := FALSE;   // CH1.Sign.Maintenance_Activated.24
   Sign.Maintenance_Activated."25" := FALSE;   // CH1.Sign.Maintenance_Activated.25
   Sign.Maintenance_Activated."26" := FALSE;   // CH1.Sign.Maintenance_Activated.26
   Sign.Maintenance_Activated."27" := FALSE;   // CH1.Sign.Maintenance_Activated.27
   Sign.Maintenance_Activated."28" := FALSE;   // CH1.Sign.Maintenance_Activated.28
   Sign.Maintenance_Activated."29" := FALSE;   // CH1.Sign.Maintenance_Activated.29
   Sign.Maintenance_Activated."30" := FALSE;   // CH1.Sign.Maintenance_Activated.30
   Sign.Maintenance_Activated."31" := FALSE;   // CH1.Sign.Maintenance_Activated.31
   Input.StaPbt := FALSE;
   Input.StoPbt := FALSE;
   Input.RstPbt := FALSE;
   Input.EnaPbt := FALSE;
   Input.Safety.SafeZoneOk := FALSE;
   Input.Safety.SafeZone2Ok := FALSE;
   Input.Safety.SrsGrdEmgNOk := TRUE;
   Input.Safety.SrsGrdEmg2NOk := FALSE;
   Input.Safety.STO_Chain1Long := TRUE;
   Input.Safety.STO_Chain2Long := TRUE;
   Input.Safety.STO_Chain3Long := TRUE;
   Input.Safety.STO_Chain4Cross := TRUE;
   Input.Safety.STO_Chain5Long := TRUE;
   Input.Safety.STO_Chain6Long := TRUE;
   Input.Safety.STO_Chain7Long := TRUE;
   Input.Safety.STO_Chain8Cross := TRUE;
   Input.Safety.QBad_Chain1Long := FALSE;
   Input.Safety.QBad_Chain2Long := FALSE;
   Input.Safety.QBad_Chain3Long := FALSE;
   Input.Safety.QBad_Chain4Cross := FALSE;
   Input.Safety.QBad_Chain5Long := FALSE;
   Input.Safety.QBad_Chain6Long := FALSE;
   Input.Safety.QBad_Chain7Long := FALSE;
   Input.Safety.QBad_Chain8Cross := FALSE;
   Output.ModLgh := FALSE;
   Ons.SpeedUp := FALSE;
   Ons.StrobeMould := TRUE;
   Ons._2 := FALSE;
   Ons._3 := FALSE;
   Ons._4 := FALSE;
   Ons._5 := FALSE;
   Ons._6 := FALSE;
   Ons._7 := FALSE;
   Ons._8 := FALSE;
   Ons._9 := FALSE;
   Ons._10 := FALSE;
   Ons._11 := FALSE;
   Ons._12 := FALSE;
   Ons._13 := FALSE;
   Ons._14 := FALSE;
   Ons._15 := FALSE;
   "Step"._00_StartLongChainWork := TRUE;
   "Step"._10_LongChainInMotion := TRUE;
   "Step"._20_AdvanceCheckStartCrossWork := FALSE;
   "Step"._30_LongChainWorkDone := FALSE;
   "Step"._40_StartCrossChainWork := FALSE;
   "Step"._50_CrossChainInMotion := FALSE;
   "Step"._60_AdvanceCheckStartLongWork := FALSE;
   "Step".ScSeqOk := FALSE;
   CamCalc.CalcReq := FALSE;
   CamCalc.LongChain_CalcReq := FALSE;
   CamCalc.CrossChain_CalcReq := FALSE;
   CamCalc.ContChain_CalcReq := FALSE;
   CamCalc.TransferChain_CalcReq := FALSE;
   CamCalc.ColumnAscChain_CalcReq := FALSE;
   CamCalc.ColumnDescChain_CalcReq := FALSE;
   CamCalc.CrossChain4_CalcReq := FALSE;
   CamCalc.OnsCalcReq := FALSE;
   CamCalc.LongChain_OnsCalcReq := FALSE;
   CamCalc.CrossChain_OnsCalcReq := FALSE;
   CamCalc.ContChain_OnsCalcReq := FALSE;
   CamCalc.TransferChain_OnsCalcReq := FALSE;
   CamCalc.ColumnAscChain_OnsCalcReq := FALSE;
   CamCalc.ColumnDescChain_OnsCalcReq := FALSE;
   CamCalc.InletCrowding_OnsCalcReq := FALSE;
   CamCalc.CrossChain4_OnsCalcReq := FALSE;
   CamCalc.LongChain_IndexProfile := 0;
   CamCalc.LongChain_LenghtUsed := 2;
   CamCalc.CrossChain_IndexProfile := 0;
   CamCalc.CrossChain_LenghtUsed := 6;
   CamCalc.ContChain_IndexProfile := 0;
   CamCalc.ContChain_LenghtUsed := 1;
   CamCalc.TransferChain_IndexProfile := 0;
   CamCalc.TransferChain_LenghtUsed := 0;
   CamCalc.ColumnAscChain_IndexProfile := 0;
   CamCalc.ColumnAscChain_LenghtUsed := 0;
   CamCalc.ColumnDescChain_IndexProfile := 0;
   CamCalc.ColumnDescChain_LenghtUsed := 0;
   CamCalc.CrossChain4_IndexProfile := 0;
   CamCalc.CrossChain4_LenghtUsed := 6;
   CamCalc.LongChain_Slope := 0.0;
   CamCalc.CrossChain_Slope := 0.0;
   CamCalc.BeltChain_Slope := 0.0;
   CamCalc.ContChain_Slope := 0.0;
   CamCalc.TransferChain_Slope := 0.0;
   CamCalc.ColumnAscChain_Slope := 0.0;
   CamCalc.ColumnDescChain_Slope := 0.0;
   CamCalc.InletCrowding_Slope := 0.0;
   CamCalc.OutletCrowding_Slope := 0.0;
   CamCalc.CrossChain4_Slope := 0.0;
   CamCalc.LongChain_Unwind := 406.4;
   CamCalc.CrossChain_Unwind := 711.2;
   CamCalc.BeltChain_Unwind := 406.4;
   CamCalc.ContChain_Unwind := 406.4;
   CamCalc.TransferChain_Unwind := 812.8;
   CamCalc.TransferChain_RevDirection := 0.0;
   CamCalc.TransferChain_Step := 812.8;
   CamCalc.ColumnAscChain_Unwind := 57.15;
   CamCalc.ColumnDescChain_Unwind := 57.15;
   CamCalc.CrossChain4_Unwind := 812.8;
   CamCalc.LongChain_Cam[0].leadingValueStart := 0.0;
   CamCalc.LongChain_Cam[1].leadingValueStart := 162.0;
   CamCalc.LongChain_Cam[2..99].leadingValueStart := 0.0;
   CamCalc.LongChain_Cam[0].leadingValueEnd := 162.0;
   CamCalc.LongChain_Cam[1].leadingValueEnd := 360.0;
   CamCalc.LongChain_Cam[2..99].leadingValueEnd := 0.0;
   CamCalc.LongChain_Cam[0].followingValueStart := 0.0;
   CamCalc.LongChain_Cam[1].followingValueStart := 406.399993896484;
   CamCalc.LongChain_Cam[2..99].followingValueStart := 0.0;
   CamCalc.LongChain_Cam[0..1].followingValueEnd := 406.399993896484;
   CamCalc.LongChain_Cam[2..99].followingValueEnd := 0.0;
   CamCalc.LongChain_Cam[0..99].geoVeloStart := 0.0;
   CamCalc.LongChain_Cam[0..99].geoVeloEnd := 0.0;
   CamCalc.LongChain_Cam[0..99].geoAccelStart := 0.0;
   CamCalc.LongChain_Cam[0..99].geoAccelEnd := 0.0;
   CamCalc.LongChain_Cam[0..99].geoJerkStart := 0.0;
   CamCalc.LongChain_Cam[0..99].geoJerkEnd := 0.0;
   CamCalc.LongChain_Cam[0..99].inflectionPointParameter := 0.5;
   CamCalc.LongChain_Cam[0..99].modVeloTrapezoidParameter := 1.0;
   CamCalc.LongChain_Cam[0..99].modSineMaxAccelCaStar := 0.0;
   CamCalc.LongChain_Cam[0].camProfileType := 5;
   CamCalc.LongChain_Cam[1].camProfileType := 2;
   CamCalc.LongChain_Cam[2..99].camProfileType := 0;
   CamCalc.CrossChain_Cam[0].leadingValueStart := 0.0;
   CamCalc.CrossChain_Cam[1].leadingValueStart := 193.679992675781;
   CamCalc.CrossChain_Cam[2..3].leadingValueStart := 225.360000610352;
   CamCalc.CrossChain_Cam[4].leadingValueStart := 328.320007324219;
   CamCalc.CrossChain_Cam[5].leadingValueStart := 360.0;
   CamCalc.CrossChain_Cam[6..99].leadingValueStart := 0.0;
   CamCalc.CrossChain_Cam[0].leadingValueEnd := 162.0;
   CamCalc.CrossChain_Cam[1..2].leadingValueEnd := 0.0;
   CamCalc.CrossChain_Cam[3].leadingValueEnd := 296.640014648438;
   CamCalc.CrossChain_Cam[4..99].leadingValueEnd := 0.0;
   CamCalc.CrossChain_Cam[0].followingValueStart := 0.0;
   CamCalc.CrossChain_Cam[1].followingValueStart := 27.8901958465576;
   CamCalc.CrossChain_Cam[2..3].followingValueStart := 167.341171264648;
   CamCalc.CrossChain_Cam[4].followingValueStart := 683.309753417969;
   CamCalc.CrossChain_Cam[5].followingValueStart := 711.200012207031;
   CamCalc.CrossChain_Cam[6..99].followingValueStart := 0.0;
   CamCalc.CrossChain_Cam[0..2].followingValueEnd := 0.0;
   CamCalc.CrossChain_Cam[3].followingValueEnd := 543.858825683594;
   CamCalc.CrossChain_Cam[4..99].followingValueEnd := 0.0;
   CamCalc.CrossChain_Cam[0..99].geoVeloStart := 0.0;
   CamCalc.CrossChain_Cam[0..99].geoVeloEnd := 0.0;
   CamCalc.CrossChain_Cam[0..99].geoAccelStart := 0.0;
   CamCalc.CrossChain_Cam[0..99].geoAccelEnd := 0.0;
   CamCalc.CrossChain_Cam[0..99].geoJerkStart := 0.0;
   CamCalc.CrossChain_Cam[0..99].geoJerkEnd := 0.0;
